LIN {X 18.143,Y -25.308,Z -49.954,A -90.000,B 90.000,C 0.000} C_DIS
LIN {X 18.670,Y -25.308,Z -49.551,A -90.000,B 90.000,C 0.000} C_DIS
LIN {X 18.953,Y -25.308,Z -49.343,A -90.000,B 90.000,C 0.000} C_DIS
LIN {X 19.482,Y -25.308,Z -48.976,A -90.000,B 90.000,C 0.000} C_DIS
LIN {X 19.664,Y -25.308,Z -48.848,A -90.000,B 90.000,C 0.000} C_DIS
LIN {X 20.308,Y -25.308,Z -48.429,A -90.000,B 90.000,C 0.000} C_DIS
LIN {X 20.824,Y -25.308,Z -48.139,A -90.000,B 90.000,C 0.000} C_DIS
LIN {X 21.214,Y -25.308,Z -47.885,A -90.000,B 90.000,C 0.000} C_DIS
LIN {X 21.722,Y -25.308,Z -47.610,A -90.000,B 90.000,C 0.000} C_DIS
LIN {X 22.049,Y -25.308,Z -47.442,A -90.000,B 90.000,C 0.000} C_DIS
LIN {X 22.838,Y -25.308,Z -47.072,A -90.000,B 90.000,C 0.000} C_DIS
LIN {X 23.297,Y -25.308,Z -46.836,A -90.000,B 90.000,C 0.000} C_DIS
LIN {X 23.748,Y -25.308,Z -46.617,A -90.000,B 90.000,C 0.000} C_DIS
LIN {X 24.114,Y -25.308,Z -46.450,A -90.000,B 90.000,C 0.000} C_DIS
LIN {X 24.501,Y -25.308,Z -46.297,A -90.000,B 90.000,C 0.000} C_DIS
LIN {X 25.566,Y -25.308,Z -45.827,A -90.000,B 90.000,C 0.000} C_DIS
LIN {X 26.230,Y -25.308,Z -45.591,A -90.000,B 90.000,C 0.000} C_DIS
LIN {X 26.539,Y -25.308,Z -45.462,A -90.000,B 90.000,C 0.000} C_DIS
LIN {X 27.063,Y -25.308,Z -45.267,A -90.000,B 90.000,C 0.000} C_DIS
LIN {X 27.873,Y -25.308,Z -45.015,A -90.000,B 90.000,C 0.000} C_DIS
LIN {X 28.137,Y -25.308,Z -44.933,A -90.000,B 90.000,C 0.000} C_DIS
LIN {X 28.312,Y -25.308,Z -44.875,A -90.000,B 90.000,C 0.000} C_DIS
LIN {X 28.933,Y -25.308,Z -44.707,A -90.000,B 90.000,C 0.000} C_DIS
LIN {X 29.591,Y -25.308,Z -44.529,A -90.000,B 90.000,C 0.000} C_DIS
LIN {X 30.404,Y -25.308,Z -44.390,A -90.000,B 90.000,C 0.000} C_DIS
LIN {X 30.883,Y -25.308,Z -44.298,A -90.000,B 90.000,C 0.000} C_DIS
LIN {X 31.361,Y -25.308,Z -44.231,A -90.000,B 90.000,C 0.000} C_DIS
LIN {X 31.445,Y -25.308,Z -44.222,A -90.000,B 90.000,C 0.000} C_DIS
LIN {X 31.957,Y -25.308,Z -44.139,A -90.000,B 90.000,C 0.000} C_DIS
LIN {X 32.533,Y -25.308,Z -44.081,A -90.000,B 90.000,C 0.000} C_DIS
LIN {X 32.602,Y -25.308,Z -44.069,A -90.000,B 90.000,C 0.000} C_DIS
LIN {X 33.150,Y -25.308,Z -43.994,A -90.000,B 90.000,C 0.000} C_DIS
LIN {X 33.474,Y -25.308,Z -43.910,A -90.000,B 90.000,C 0.000} C_DIS
LIN {X 34.801,Y -25.308,Z -43.463,A -90.000,B 90.000,C 0.000} C_DIS
LIN {X 36.507,Y -25.308,Z -42.820,A -90.000,B 90.000,C 0.000} C_DIS
LIN {X 38.163,Y -25.308,Z -42.257,A -90.000,B 90.000,C 0.000} C_DIS
LIN {X 38.421,Y -25.308,Z -42.166,A -90.000,B 90.000,C 0.000} C_DIS
LIN {X 38.842,Y -25.308,Z -42.036,A -90.000,B 90.000,C 0.000} C_DIS
LIN {X 38.933,Y -25.308,Z -42.009,A -90.000,B 90.000,C 0.000} C_DIS
LIN {X 40.215,Y -25.308,Z -41.708,A -90.000,B 90.000,C 0.000} C_DIS
LIN {X 40.698,Y -25.308,Z -41.598,A -90.000,B 90.000,C 0.000} C_DIS
LIN {X 41.808,Y -25.308,Z -41.425,A -90.000,B 90.000,C 0.000} C_DIS
LIN {X 42.260,Y -25.308,Z -41.365,A -90.000,B 90.000,C 0.000} C_DIS
LIN {X 42.548,Y -25.308,Z -41.331,A -90.000,B 90.000,C 0.000} C_DIS
LIN {X 42.938,Y -25.308,Z -41.302,A -90.000,B 90.000,C 0.000} C_DIS
LIN {X 43.127,Y -25.308,Z -41.298,A -90.000,B 90.000,C 0.000} C_DIS
LIN {X 44.357,Y -25.308,Z -41.301,A -90.000,B 90.000,C 0.000} C_DIS
LIN {X 44.824,Y -25.308,Z -41.310,A -90.000,B 90.000,C 0.000} C_DIS
LIN {X 46.077,Y -25.308,Z -41.438,A -90.000,B 90.000,C 0.000} C_DIS
LIN {X 46.591,Y -25.308,Z -41.498,A -90.000,B 90.000,C 0.000} C_DIS
LIN {X 46.783,Y -25.308,Z -41.522,A -90.000,B 90.000,C 0.000} C_DIS
LIN {X 47.059,Y -25.308,Z -41.565,A -90.000,B 90.000,C 0.000} C_DIS
LIN {X 47.466,Y -25.308,Z -41.664,A -90.000,B 90.000,C 0.000} C_DIS
LIN {X 47.871,Y -25.308,Z -41.771,A -90.000,B 90.000,C 0.000} C_DIS
LIN {X 49.147,Y -25.308,Z -42.145,A -90.000,B 90.000,C 0.000} C_DIS
LIN {X 50.476,Y -25.308,Z -42.617,A -90.000,B 90.000,C 0.000} C_DIS
LIN {X 50.921,Y -25.308,Z -42.786,A -90.000,B 90.000,C 0.000} C_DIS
LIN {X 51.227,Y -25.308,Z -42.923,A -90.000,B 90.000,C 0.000} C_DIS
LIN {X 52.706,Y -25.308,Z -43.641,A -90.000,B 90.000,C 0.000} C_DIS
LIN {X 53.133,Y -25.308,Z -43.865,A -90.000,B 90.000,C 0.000} C_DIS
LIN {X 53.694,Y -25.308,Z -44.165,A -90.000,B 90.000,C 0.000} C_DIS
LIN {X 54.079,Y -25.308,Z -44.378,A -90.000,B 90.000,C 0.000} C_DIS
LIN {X 54.481,Y -25.308,Z -44.646,A -90.000,B 90.000,C 0.000} C_DIS
LIN {X 55.761,Y -25.308,Z -45.510,A -90.000,B 90.000,C 0.000} C_DIS
LIN {X 56.981,Y -25.308,Z -46.342,A -90.000,B 90.000,C 0.000} C_DIS
LIN {X 57.354,Y -25.308,Z -46.650,A -90.000,B 90.000,C 0.000} C_DIS
LIN {X 59.159,Y -25.308,Z -48.157,A -90.000,B 90.000,C 0.000} C_DIS
LIN {X 59.556,Y -25.308,Z -48.497,A -90.000,B 90.000,C 0.000} C_DIS
LIN {X 61.541,Y -25.308,Z -50.392,A -90.000,B 90.000,C 0.000} C_DIS
LIN {X 62.293,Y -25.308,Z -51.104,A -90.000,B 90.000,C 0.000} C_DIS
LIN {X 63.430,Y -25.308,Z -52.202,A -90.000,B 90.000,C 0.000} C_DIS
LIN {X 64.564,Y -25.308,Z -53.172,A -90.000,B 90.000,C 0.000} C_DIS
LIN {X 65.147,Y -25.308,Z -53.687,A -90.000,B 90.000,C 0.000} C_DIS
LIN {X 65.829,Y -25.308,Z -54.185,A -90.000,B 90.000,C 0.000} C_DIS
LIN {X 67.069,Y -25.308,Z -55.053,A -90.000,B 90.000,C 0.000} C_DIS
LIN {X 67.323,Y -25.308,Z -55.221,A -90.000,B 90.000,C 0.000} C_DIS
LIN {X 68.793,Y -25.308,Z -56.153,A -90.000,B 90.000,C 0.000} C_DIS
LIN {X 69.363,Y -25.308,Z -56.519,A -90.000,B 90.000,C 0.000} C_DIS
LIN {X 70.905,Y -25.308,Z -57.502,A -90.000,B 90.000,C 0.000} C_DIS
LIN {X 71.252,Y -25.308,Z -57.727,A -90.000,B 90.000,C 0.000} C_DIS
LIN {X 71.570,Y -25.308,Z -57.963,A -90.000,B 90.000,C 0.000} C_DIS
LIN {X 73.123,Y -25.308,Z -59.076,A -90.000,B 90.000,C 0.000} C_DIS
LIN {X 73.494,Y -25.308,Z -59.375,A -90.000,B 90.000,C 0.000} C_DIS
LIN {X 74.370,Y -25.308,Z -60.174,A -90.000,B 90.000,C 0.000} C_DIS
LIN {X 75.025,Y -25.308,Z -60.802,A -90.000,B 90.000,C 0.000} C_DIS
LIN {X 75.362,Y -25.308,Z -61.138,A -90.000,B 90.000,C 0.000} C_DIS
LIN {X 75.788,Y -25.308,Z -61.621,A -90.000,B 90.000,C 0.000} C_DIS
LIN {X 76.413,Y -25.308,Z -62.367,A -90.000,B 90.000,C 0.000} C_DIS
LIN {X 76.829,Y -25.308,Z -62.865,A -90.000,B 90.000,C 0.000} C_DIS
LIN {X 77.271,Y -25.308,Z -63.464,A -90.000,B 90.000,C 0.000} C_DIS
LIN {X 77.867,Y -25.308,Z -64.321,A -90.000,B 90.000,C 0.000} C_DIS
LIN {X 78.264,Y -25.308,Z -64.917,A -90.000,B 90.000,C 0.000} C_DIS
LIN {X 78.540,Y -25.308,Z -65.359,A -90.000,B 90.000,C 0.000} C_DIS
LIN {X 79.035,Y -25.308,Z -63.677,A -90.000,B 90.000,C 0.000} C_DIS
LIN {X 79.744,Y -25.308,Z -61.550,A -90.000,B 90.000,C 0.000} C_DIS
LIN {X 79.787,Y -25.308,Z -61.436,A -90.000,B 90.000,C 0.000} C_DIS
LIN {X 80.298,Y -25.308,Z -59.798,A -90.000,B 90.000,C 0.000} C_DIS
LIN {X 80.453,Y -25.308,Z -59.335,A -90.000,B 90.000,C 0.000} C_DIS
LIN {X 81.205,Y -25.308,Z -57.294,A -90.000,B 90.000,C 0.000} C_DIS
LIN {X 81.746,Y -25.308,Z -56.077,A -90.000,B 90.000,C 0.000} C_DIS
LIN {X 82.134,Y -25.308,Z -55.110,A -90.000,B 90.000,C 0.000} C_DIS
LIN {X 82.335,Y -25.308,Z -54.666,A -90.000,B 90.000,C 0.000} C_DIS
LIN {X 83.333,Y -25.308,Z -52.807,A -90.000,B 90.000,C 0.000} C_DIS
LIN {X 83.579,Y -25.308,Z -52.386,A -90.000,B 90.000,C 0.000} C_DIS
LIN {X 84.744,Y -25.308,Z -50.676,A -90.000,B 90.000,C 0.000} C_DIS
LIN {X 85.030,Y -25.308,Z -50.284,A -90.000,B 90.000,C 0.000} C_DIS
LIN {X 86.347,Y -25.308,Z -48.703,A -90.000,B 90.000,C 0.000} C_DIS
LIN {X 86.674,Y -25.308,Z -48.341,A -90.000,B 90.000,C 0.000} C_DIS
LIN {X 88.117,Y -25.308,Z -46.880,A -90.000,B 90.000,C 0.000} C_DIS
LIN {X 88.495,Y -25.308,Z -46.539,A -90.000,B 90.000,C 0.000} C_DIS
LIN {X 90.061,Y -25.308,Z -45.164,A -90.000,B 90.000,C 0.000} C_DIS
LIN {X 91.724,Y -25.308,Z -43.871,A -90.000,B 90.000,C 0.000} C_DIS
LIN {X 92.141,Y -25.308,Z -43.566,A -90.000,B 90.000,C 0.000} C_DIS
LIN {X 93.780,Y -25.308,Z -42.419,A -90.000,B 90.000,C 0.000} C_DIS
LIN {X 95.430,Y -25.308,Z -41.375,A -90.000,B 90.000,C 0.000} C_DIS
LIN {X 95.885,Y -25.308,Z -41.109,A -90.000,B 90.000,C 0.000} C_DIS
LIN {X 97.376,Y -25.308,Z -40.260,A -90.000,B 90.000,C 0.000} C_DIS
LIN {X 98.805,Y -25.308,Z -39.523,A -90.000,B 90.000,C 0.000} C_DIS
LIN {X 100.339,Y -25.308,Z -38.797,A -90.000,B 90.000,C 0.000} C_DIS
LIN {X 102.099,Y -25.308,Z -37.999,A -90.000,B 90.000,C 0.000} C_DIS
LIN {X 103.528,Y -25.308,Z -37.362,A -90.000,B 90.000,C 0.000} C_DIS
LIN {X 104.529,Y -25.308,Z -36.920,A -90.000,B 90.000,C 0.000} C_DIS
LIN {X 105.418,Y -25.308,Z -36.546,A -90.000,B 90.000,C 0.000} C_DIS
LIN {X 106.878,Y -25.308,Z -35.966,A -90.000,B 90.000,C 0.000} C_DIS
LIN {X 107.402,Y -25.308,Z -35.767,A -90.000,B 90.000,C 0.000} C_DIS
LIN {X 107.855,Y -25.308,Z -35.604,A -90.000,B 90.000,C 0.000} C_DIS
LIN {X 108.317,Y -25.308,Z -35.448,A -90.000,B 90.000,C 0.000} C_DIS
LIN {X 108.777,Y -25.308,Z -35.326,A -90.000,B 90.000,C 0.000} C_DIS
LIN {X 109.221,Y -25.308,Z -35.225,A -90.000,B 90.000,C 0.000} C_DIS
LIN {X 109.760,Y -25.308,Z -35.155,A -90.000,B 90.000,C 0.000} C_DIS
LIN {X 110.108,Y -25.308,Z -35.113,A -90.000,B 90.000,C 0.000} C_DIS
LIN {X 110.563,Y -25.308,Z -35.105,A -90.000,B 90.000,C 0.000} C_DIS
LIN {X 110.619,Y -25.308,Z -35.106,A -90.000,B 90.000,C 0.000} C_DIS
LIN {X 110.949,Y -25.308,Z -35.117,A -90.000,B 90.000,C 0.000} C_DIS
LIN {X 111.445,Y -25.308,Z -35.160,A -90.000,B 90.000,C 0.000} C_DIS
LIN {X 112.068,Y -25.308,Z -35.277,A -90.000,B 90.000,C 0.000} C_DIS
LIN {X 112.405,Y -25.308,Z -35.362,A -90.000,B 90.000,C 0.000} C_DIS
LIN {X 112.925,Y -25.308,Z -35.518,A -90.000,B 90.000,C 0.000} C_DIS
LIN {X 113.055,Y -25.308,Z -35.560,A -90.000,B 90.000,C 0.000} C_DIS
LIN {X 113.505,Y -25.308,Z -35.746,A -90.000,B 90.000,C 0.000} C_DIS
LIN {X 113.979,Y -25.308,Z -35.973,A -90.000,B 90.000,C 0.000} C_DIS
LIN {X 114.418,Y -25.308,Z -36.210,A -90.000,B 90.000,C 0.000} C_DIS
LIN {X 114.540,Y -25.308,Z -36.286,A -90.000,B 90.000,C 0.000} C_DIS
LIN {X 114.952,Y -25.308,Z -36.566,A -90.000,B 90.000,C 0.000} C_DIS
LIN {X 115.050,Y -25.308,Z -36.644,A -90.000,B 90.000,C 0.000} C_DIS
LIN {X 115.450,Y -25.308,Z -36.982,A -90.000,B 90.000,C 0.000} C_DIS
LIN {X 115.513,Y -25.308,Z -37.039,A -90.000,B 90.000,C 0.000} C_DIS
LIN {X 115.921,Y -25.308,Z -37.462,A -90.000,B 90.000,C 0.000} C_DIS
LIN {X 116.080,Y -25.308,Z -37.632,A -90.000,B 90.000,C 0.000} C_DIS
LIN {X 116.439,Y -25.308,Z -38.088,A -90.000,B 90.000,C 0.000} C_DIS
LIN {X 116.700,Y -25.308,Z -38.500,A -90.000,B 90.000,C 0.000} C_DIS
LIN {X 116.928,Y -25.308,Z -38.961,A -90.000,B 90.000,C 0.000} C_DIS
LIN {X 117.066,Y -25.308,Z -39.268,A -90.000,B 90.000,C 0.000} C_DIS
LIN {X 117.142,Y -25.308,Z -39.466,A -90.000,B 90.000,C 0.000} C_DIS
LIN {X 117.260,Y -25.308,Z -39.781,A -90.000,B 90.000,C 0.000} C_DIS
LIN {X 117.390,Y -25.308,Z -40.280,A -90.000,B 90.000,C 0.000} C_DIS
LIN {X 117.462,Y -25.308,Z -40.593,A -90.000,B 90.000,C 0.000} C_DIS
LIN {X 117.541,Y -25.308,Z -41.107,A -90.000,B 90.000,C 0.000} C_DIS
LIN {X 117.596,Y -25.308,Z -41.523,A -90.000,B 90.000,C 0.000} C_DIS
LIN {X 117.630,Y -25.308,Z -41.874,A -90.000,B 90.000,C 0.000} C_DIS
LIN {X 117.659,Y -25.308,Z -42.461,A -90.000,B 90.000,C 0.000} C_DIS
LIN {X 117.668,Y -25.308,Z -42.696,A -90.000,B 90.000,C 0.000} C_DIS
LIN {X 117.664,Y -25.308,Z -42.866,A -90.000,B 90.000,C 0.000} C_DIS
LIN {X 117.661,Y -25.308,Z -42.950,A -90.000,B 90.000,C 0.000} C_DIS
LIN {X 117.651,Y -25.308,Z -43.202,A -90.000,B 90.000,C 0.000} C_DIS
LIN {X 117.607,Y -25.308,Z -43.721,A -90.000,B 90.000,C 0.000} C_DIS
LIN {X 117.567,Y -25.308,Z -44.117,A -90.000,B 90.000,C 0.000} C_DIS
LIN {X 117.482,Y -25.308,Z -44.670,A -90.000,B 90.000,C 0.000} C_DIS
LIN {X 117.399,Y -25.308,Z -45.114,A -90.000,B 90.000,C 0.000} C_DIS
LIN {X 117.260,Y -25.308,Z -45.739,A -90.000,B 90.000,C 0.000} C_DIS
LIN {X 117.105,Y -25.308,Z -46.261,A -90.000,B 90.000,C 0.000} C_DIS
LIN {X 116.900,Y -25.308,Z -46.938,A -90.000,B 90.000,C 0.000} C_DIS
LIN {X 116.546,Y -25.308,Z -47.857,A -90.000,B 90.000,C 0.000} C_DIS
LIN {X 116.372,Y -25.308,Z -48.278,A -90.000,B 90.000,C 0.000} C_DIS
LIN {X 115.873,Y -25.308,Z -49.350,A -90.000,B 90.000,C 0.000} C_DIS
LIN {X 115.235,Y -25.308,Z -50.626,A -90.000,B 90.000,C 0.000} C_DIS
LIN {X 114.577,Y -25.308,Z -51.931,A -90.000,B 90.000,C 0.000} C_DIS
LIN {X 113.941,Y -25.308,Z -53.229,A -90.000,B 90.000,C 0.000} C_DIS
LIN {X 113.276,Y -25.308,Z -54.687,A -90.000,B 90.000,C 0.000} C_DIS
LIN {X 112.799,Y -25.308,Z -55.830,A -90.000,B 90.000,C 0.000} C_DIS
LIN {X 112.213,Y -25.308,Z -57.388,A -90.000,B 90.000,C 0.000} C_DIS
LIN {X 111.674,Y -25.308,Z -59.009,A -90.000,B 90.000,C 0.000} C_DIS
LIN {X 111.260,Y -25.308,Z -60.445,A -90.000,B 90.000,C 0.000} C_DIS
LIN {X 110.703,Y -25.308,Z -62.486,A -90.000,B 90.000,C 0.000} C_DIS
LIN {X 110.152,Y -25.308,Z -64.437,A -90.000,B 90.000,C 0.000} C_DIS
LIN {X 110.021,Y -25.308,Z -64.879,A -90.000,B 90.000,C 0.000} C_DIS
LIN {X 109.345,Y -25.308,Z -67.050,A -90.000,B 90.000,C 0.000} C_DIS
LIN {X 108.519,Y -25.308,Z -69.358,A -90.000,B 90.000,C 0.000} C_DIS
LIN {X 107.550,Y -25.308,Z -71.793,A -90.000,B 90.000,C 0.000} C_DIS
LIN {X 107.403,Y -25.308,Z -72.150,A -90.000,B 90.000,C 0.000} C_DIS
LIN {X 106.414,Y -25.308,Z -74.420,A -90.000,B 90.000,C 0.000} C_DIS
LIN {X 105.411,Y -25.308,Z -76.516,A -90.000,B 90.000,C 0.000} C_DIS
LIN {X 104.209,Y -25.308,Z -78.763,A -90.000,B 90.000,C 0.000} C_DIS
LIN {X 103.943,Y -25.308,Z -79.223,A -90.000,B 90.000,C 0.000} C_DIS
LIN {X 103.058,Y -25.308,Z -80.726,A -90.000,B 90.000,C 0.000} C_DIS
LIN {X 102.880,Y -25.308,Z -81.006,A -90.000,B 90.000,C 0.000} C_DIS
LIN {X 102.164,Y -25.308,Z -82.128,A -90.000,B 90.000,C 0.000} C_DIS
LIN {X 99.737,Y -25.308,Z -85.762,A -90.000,B 90.000,C 0.000} C_DIS
LIN {X 99.776,Y -25.308,Z -86.269,A -90.000,B 90.000,C 0.000} C_DIS
LIN {X 99.848,Y -25.308,Z -87.593,A -90.000,B 90.000,C 0.000} C_DIS
LIN {X 99.953,Y -25.308,Z -88.797,A -90.000,B 90.000,C 0.000} C_DIS
LIN {X 99.978,Y -25.308,Z -89.273,A -90.000,B 90.000,C 0.000} C_DIS
LIN {X 99.997,Y -25.308,Z -89.800,A -90.000,B 90.000,C 0.000} C_DIS
LIN {X 100.015,Y -25.308,Z -90.712,A -90.000,B 90.000,C 0.000} C_DIS
LIN {X 100.028,Y -25.308,Z -91.629,A -90.000,B 90.000,C 0.000} C_DIS
LIN {X 100.042,Y -25.308,Z -92.081,A -90.000,B 90.000,C 0.000} C_DIS
LIN {X 100.041,Y -25.308,Z -92.155,A -90.000,B 90.000,C 0.000} C_DIS
LIN {X 99.990,Y -25.308,Z -93.020,A -90.000,B 90.000,C 0.000} C_DIS
LIN {X 99.954,Y -25.308,Z -93.959,A -90.000,B 90.000,C 0.000} C_DIS
LIN {X 99.931,Y -25.308,Z -94.384,A -90.000,B 90.000,C 0.000} C_DIS
LIN {X 99.913,Y -25.308,Z -94.531,A -90.000,B 90.000,C 0.000} C_DIS
LIN {X 99.819,Y -25.308,Z -95.415,A -90.000,B 90.000,C 0.000} C_DIS
LIN {X 99.799,Y -25.308,Z -95.920,A -90.000,B 90.000,C 0.000} C_DIS
LIN {X 99.741,Y -25.308,Z -96.399,A -90.000,B 90.000,C 0.000} C_DIS
LIN {X 99.696,Y -25.308,Z -96.658,A -90.000,B 90.000,C 0.000} C_DIS
LIN {X 99.644,Y -25.308,Z -97.627,A -90.000,B 90.000,C 0.000} C_DIS
LIN {X 99.544,Y -25.308,Z -99.179,A -90.000,B 90.000,C 0.000} C_DIS
LIN {X 99.527,Y -25.308,Z -99.300,A -90.000,B 90.000,C 0.000} C_DIS
LIN {X 99.435,Y -25.308,Z -100.699,A -90.000,B 90.000,C 0.000} C_DIS
LIN {X 99.398,Y -25.308,Z -100.988,A -90.000,B 90.000,C 0.000} C_DIS
LIN {X 99.340,Y -25.308,Z -102.329,A -90.000,B 90.000,C 0.000} C_DIS
LIN {X 99.327,Y -25.308,Z -102.468,A -90.000,B 90.000,C 0.000} C_DIS
LIN {X 99.324,Y -25.308,Z -103.358,A -90.000,B 90.000,C 0.000} C_DIS
LIN {X 99.312,Y -25.308,Z -103.683,A -90.000,B 90.000,C 0.000} C_DIS
LIN {X 99.307,Y -25.308,Z -103.795,A -90.000,B 90.000,C 0.000} C_DIS
LIN {X 99.321,Y -25.308,Z -104.026,A -90.000,B 90.000,C 0.000} C_DIS
LIN {X 99.361,Y -25.308,Z -104.573,A -90.000,B 90.000,C 0.000} C_DIS
LIN {X 99.427,Y -25.308,Z -105.073,A -90.000,B 90.000,C 0.000} C_DIS
LIN {X 99.488,Y -25.308,Z -105.508,A -90.000,B 90.000,C 0.000} C_DIS
LIN {X 99.631,Y -25.308,Z -106.321,A -90.000,B 90.000,C 0.000} C_DIS
LIN {X 99.899,Y -25.308,Z -107.995,A -90.000,B 90.000,C 0.000} C_DIS
LIN {X 99.981,Y -25.308,Z -108.804,A -90.000,B 90.000,C 0.000} C_DIS
LIN {X 100.053,Y -25.308,Z -109.443,A -90.000,B 90.000,C 0.000} C_DIS
LIN {X 100.126,Y -25.308,Z -110.453,A -90.000,B 90.000,C 0.000} C_DIS
LIN {X 100.183,Y -25.308,Z -111.111,A -90.000,B 90.000,C 0.000} C_DIS
LIN {X 100.229,Y -25.308,Z -111.892,A -90.000,B 90.000,C 0.000} C_DIS
LIN {X 100.310,Y -25.308,Z -112.963,A -90.000,B 90.000,C 0.000} C_DIS
LIN {X 100.359,Y -25.308,Z -113.831,A -90.000,B 90.000,C 0.000} C_DIS
LIN {X 100.445,Y -25.308,Z -115.019,A -90.000,B 90.000,C 0.000} C_DIS
LIN {X 100.533,Y -25.308,Z -116.130,A -90.000,B 90.000,C 0.000} C_DIS
LIN {X 100.601,Y -25.308,Z -117.246,A -90.000,B 90.000,C 0.000} C_DIS
LIN {X 100.674,Y -25.308,Z -118.213,A -90.000,B 90.000,C 0.000} C_DIS
LIN {X 100.751,Y -25.308,Z -119.583,A -90.000,B 90.000,C 0.000} C_DIS
LIN {X 100.800,Y -25.308,Z -120.356,A -90.000,B 90.000,C 0.000} C_DIS
LIN {X 100.825,Y -25.308,Z -120.811,A -90.000,B 90.000,C 0.000} C_DIS
LIN {X 100.921,Y -25.308,Z -122.978,A -90.000,B 90.000,C 0.000} C_DIS
LIN {X 100.945,Y -25.308,Z -123.620,A -90.000,B 90.000,C 0.000} C_DIS
LIN {X 100.973,Y -25.308,Z -124.815,A -90.000,B 90.000,C 0.000} C_DIS
LIN {X 100.968,Y -25.308,Z -126.202,A -90.000,B 90.000,C 0.000} C_DIS
LIN {X 100.978,Y -25.308,Z -127.131,A -90.000,B 90.000,C 0.000} C_DIS
LIN {X 100.927,Y -25.308,Z -128.864,A -90.000,B 90.000,C 0.000} C_DIS
LIN {X 100.912,Y -25.308,Z -129.693,A -90.000,B 90.000,C 0.000} C_DIS
LIN {X 100.815,Y -25.308,Z -131.616,A -90.000,B 90.000,C 0.000} C_DIS
LIN {X 100.792,Y -25.308,Z -132.231,A -90.000,B 90.000,C 0.000} C_DIS
LIN {X 100.655,Y -25.308,Z -134.453,A -90.000,B 90.000,C 0.000} C_DIS
LIN {X 100.615,Y -25.308,Z -135.207,A -90.000,B 90.000,C 0.000} C_DIS
LIN {X 100.584,Y -25.308,Z -135.733,A -90.000,B 90.000,C 0.000} C_DIS
LIN {X 100.370,Y -25.308,Z -138.988,A -90.000,B 90.000,C 0.000} C_DIS
LIN {X 100.175,Y -25.308,Z -141.689,A -90.000,B 90.000,C 0.000} C_DIS
LIN {X 100.021,Y -25.308,Z -143.726,A -90.000,B 90.000,C 0.000} C_DIS
LIN {X 99.864,Y -25.308,Z -145.627,A -90.000,B 90.000,C 0.000} C_DIS
LIN {X 99.651,Y -25.308,Z -148.108,A -90.000,B 90.000,C 0.000} C_DIS
LIN {X 99.528,Y -25.308,Z -149.393,A -90.000,B 90.000,C 0.000} C_DIS
LIN {X 99.410,Y -25.308,Z -150.436,A -90.000,B 90.000,C 0.000} C_DIS
LIN {X 99.155,Y -25.308,Z -153.045,A -90.000,B 90.000,C 0.000} C_DIS
LIN {X 99.077,Y -25.308,Z -153.644,A -90.000,B 90.000,C 0.000} C_DIS
LIN {X 99.058,Y -25.308,Z -153.783,A -90.000,B 90.000,C 0.000} C_DIS
LIN {X 98.742,Y -25.308,Z -156.680,A -90.000,B 90.000,C 0.000} C_DIS
LIN {X 98.709,Y -25.308,Z -156.898,A -90.000,B 90.000,C 0.000} C_DIS
LIN {X 98.400,Y -25.308,Z -159.435,A -90.000,B 90.000,C 0.000} C_DIS
LIN {X 98.332,Y -25.308,Z -160.140,A -90.000,B 90.000,C 0.000} C_DIS
LIN {X 98.002,Y -25.308,Z -162.603,A -90.000,B 90.000,C 0.000} C_DIS
LIN {X 97.876,Y -25.308,Z -163.832,A -90.000,B 90.000,C 0.000} C_DIS
LIN {X 97.601,Y -25.308,Z -165.718,A -90.000,B 90.000,C 0.000} C_DIS
LIN {X 97.397,Y -25.308,Z -167.595,A -90.000,B 90.000,C 0.000} C_DIS
LIN {X 97.263,Y -25.308,Z -168.464,A -90.000,B 90.000,C 0.000} C_DIS
LIN {X 96.949,Y -25.308,Z -171.253,A -90.000,B 90.000,C 0.000} C_DIS
LIN {X 96.874,Y -25.308,Z -171.737,A -90.000,B 90.000,C 0.000} C_DIS
LIN {X 96.488,Y -25.308,Z -175.168,A -90.000,B 90.000,C 0.000} C_DIS
LIN {X 96.182,Y -25.308,Z -177.661,A -90.000,B 90.000,C 0.000} C_DIS
LIN {X 96.152,Y -25.308,Z -177.991,A -90.000,B 90.000,C 0.000} C_DIS
LIN {X 95.896,Y -25.308,Z -180.202,A -90.000,B 90.000,C 0.000} C_DIS
LIN {X 95.835,Y -25.308,Z -180.892,A -90.000,B 90.000,C 0.000} C_DIS
LIN {X 95.662,Y -25.308,Z -182.520,A -90.000,B 90.000,C 0.000} C_DIS
LIN {X 95.576,Y -25.308,Z -183.541,A -90.000,B 90.000,C 0.000} C_DIS
LIN {X 95.467,Y -25.308,Z -184.688,A -90.000,B 90.000,C 0.000} C_DIS
LIN {X 95.336,Y -25.308,Z -186.329,A -90.000,B 90.000,C 0.000} C_DIS
LIN {X 95.306,Y -25.308,Z -186.689,A -90.000,B 90.000,C 0.000} C_DIS
LIN {X 95.191,Y -25.308,Z -188.281,A -90.000,B 90.000,C 0.000} C_DIS
LIN {X 95.023,Y -25.308,Z -190.814,A -90.000,B 90.000,C 0.000} C_DIS
LIN {X 95.011,Y -25.308,Z -190.963,A -90.000,B 90.000,C 0.000} C_DIS
LIN {X 94.740,Y -25.308,Z -193.398,A -90.000,B 90.000,C 0.000} C_DIS
LIN {X 94.454,Y -25.308,Z -195.346,A -90.000,B 90.000,C 0.000} C_DIS
LIN {X 94.234,Y -25.308,Z -196.731,A -90.000,B 90.000,C 0.000} C_DIS
LIN {X 93.663,Y -25.308,Z -199.595,A -90.000,B 90.000,C 0.000} C_DIS
LIN {X 93.542,Y -25.308,Z -200.212,A -90.000,B 90.000,C 0.000} C_DIS
LIN {X 92.828,Y -25.308,Z -203.214,A -90.000,B 90.000,C 0.000} C_DIS
LIN {X 92.544,Y -25.308,Z -204.440,A -90.000,B 90.000,C 0.000} C_DIS
LIN {X 91.801,Y -25.308,Z -207.333,A -90.000,B 90.000,C 0.000} C_DIS
LIN {X 91.325,Y -25.308,Z -209.244,A -90.000,B 90.000,C 0.000} C_DIS
LIN {X 90.642,Y -25.308,Z -211.832,A -90.000,B 90.000,C 0.000} C_DIS
LIN {X 89.972,Y -25.308,Z -214.447,A -90.000,B 90.000,C 0.000} C_DIS
LIN {X 89.411,Y -25.308,Z -216.578,A -90.000,B 90.000,C 0.000} C_DIS
LIN {X 88.171,Y -25.308,Z -221.432,A -90.000,B 90.000,C 0.000} C_DIS
LIN {X 87.204,Y -25.308,Z -225.322,A -90.000,B 90.000,C 0.000} C_DIS
LIN {X 86.940,Y -25.308,Z -226.315,A -90.000,B 90.000,C 0.000} C_DIS
LIN {X 85.743,Y -25.308,Z -230.924,A -90.000,B 90.000,C 0.000} C_DIS
LIN {X 85.646,Y -25.308,Z -231.281,A -90.000,B 90.000,C 0.000} C_DIS
LIN {X 85.522,Y -25.308,Z -231.698,A -90.000,B 90.000,C 0.000} C_DIS
LIN {X 84.416,Y -25.308,Z -235.552,A -90.000,B 90.000,C 0.000} C_DIS
LIN {X 83.986,Y -25.308,Z -237.019,A -90.000,B 90.000,C 0.000} C_DIS
LIN {X 81.908,Y -25.308,Z -243.223,A -90.000,B 90.000,C 0.000} C_DIS
LIN {X 81.778,Y -25.308,Z -243.561,A -90.000,B 90.000,C 0.000} C_DIS
LIN {X 81.778,Y -60.000,Z -243.561,A -90.000,B 90.000,C 0.000} C_DIS
LIN {X 99.796,Y -60.000,Z -86.519,A -90.000,B 90.000,C 0.000} C_DIS
LIN {X 99.796,Y -23.308,Z -86.519,A -90.000,B 90.000,C 0.000} C_DIS
LIN {X 99.871,Y -23.309,Z -87.492,A -90.000,B 90.000,C 0.000} C_DIS
LIN {X 100.033,Y -23.309,Z -89.800,A -90.000,B 90.000,C 0.000} C_DIS
LIN {X 100.049,Y -23.309,Z -90.038,A -90.000,B 90.000,C 0.000} C_DIS
LIN {X 100.093,Y -23.310,Z -90.499,A -90.000,B 90.000,C 0.000} C_DIS
LIN {X 100.109,Y -23.311,Z -90.717,A -90.000,B 90.000,C 0.000} C_DIS
LIN {X 100.173,Y -23.313,Z -91.776,A -90.000,B 90.000,C 0.000} C_DIS
LIN {X 100.205,Y -23.315,Z -92.181,A -90.000,B 90.000,C 0.000} C_DIS
LIN {X 100.234,Y -23.319,Z -92.418,A -90.000,B 90.000,C 0.000} C_DIS
LIN {X 100.259,Y -23.326,Z -92.902,A -90.000,B 90.000,C 0.000} C_DIS
LIN {X 100.244,Y -23.328,Z -93.631,A -90.000,B 90.000,C 0.000} C_DIS
LIN {X 100.269,Y -23.339,Z -94.490,A -90.000,B 90.000,C 0.000} C_DIS
LIN {X 100.271,Y -23.340,Z -94.538,A -90.000,B 90.000,C 0.000} C_DIS
LIN {X 100.259,Y -23.345,Z -94.860,A -90.000,B 90.000,C 0.000} C_DIS
LIN {X 100.222,Y -23.350,Z -95.541,A -90.000,B 90.000,C 0.000} C_DIS
LIN {X 100.217,Y -23.350,Z -95.646,A -90.000,B 90.000,C 0.000} C_DIS
LIN {X 100.224,Y -23.354,Z -95.935,A -90.000,B 90.000,C 0.000} C_DIS
LIN {X 100.212,Y -23.360,Z -96.257,A -90.000,B 90.000,C 0.000} C_DIS
LIN {X 100.177,Y -23.368,Z -96.708,A -90.000,B 90.000,C 0.000} C_DIS
LIN {X 100.162,Y -23.367,Z -96.923,A -90.000,B 90.000,C 0.000} C_DIS
LIN {X 100.162,Y -23.367,Z -96.956,A -90.000,B 90.000,C 0.000} C_DIS
LIN {X 100.164,Y -23.387,Z -98.180,A -90.000,B 90.000,C 0.000} C_DIS
LIN {X 100.163,Y -23.389,Z -98.333,A -90.000,B 90.000,C 0.000} C_DIS
LIN {X 100.144,Y -23.391,Z -98.741,A -90.000,B 90.000,C 0.000} C_DIS
LIN {X 100.124,Y -23.391,Z -99.045,A -90.000,B 90.000,C 0.000} C_DIS
LIN {X 100.126,Y -23.398,Z -99.275,A -90.000,B 90.000,C 0.000} C_DIS
LIN {X 100.129,Y -23.412,Z -99.834,A -90.000,B 90.000,C 0.000} C_DIS
LIN {X 100.110,Y -23.415,Z -100.241,A -90.000,B 90.000,C 0.000} C_DIS
LIN {X 100.081,Y -23.415,Z -100.672,A -90.000,B 90.000,C 0.000} C_DIS
LIN {X 100.086,Y -23.431,Z -101.042,A -90.000,B 90.000,C 0.000} C_DIS
LIN {X 100.092,Y -23.437,Z -101.310,A -90.000,B 90.000,C 0.000} C_DIS
LIN {X 100.065,Y -23.439,Z -102.005,A -90.000,B 90.000,C 0.000} C_DIS
LIN {X 100.057,Y -23.439,Z -102.203,A -90.000,B 90.000,C 0.000} C_DIS
LIN {X 100.069,Y -23.452,Z -102.533,A -90.000,B 90.000,C 0.000} C_DIS
LIN {X 100.088,Y -23.460,Z -102.959,A -90.000,B 90.000,C 0.000} C_DIS
LIN {X 100.086,Y -23.461,Z -103.455,A -90.000,B 90.000,C 0.000} C_DIS
LIN {X 100.086,Y -23.462,Z -103.545,A -90.000,B 90.000,C 0.000} C_DIS
LIN {X 100.103,Y -23.472,Z -103.832,A -90.000,B 90.000,C 0.000} C_DIS
LIN {X 100.116,Y -23.473,Z -103.986,A -90.000,B 90.000,C 0.000} C_DIS
LIN {X 100.166,Y -23.480,Z -104.480,A -90.000,B 90.000,C 0.000} C_DIS
LIN {X 100.256,Y -23.482,Z -105.112,A -90.000,B 90.000,C 0.000} C_DIS
LIN {X 100.300,Y -23.484,Z -105.388,A -90.000,B 90.000,C 0.000} C_DIS
LIN {X 100.456,Y -23.485,Z -106.279,A -90.000,B 90.000,C 0.000} C_DIS
LIN {X 100.723,Y -23.487,Z -107.938,A -90.000,B 90.000,C 0.000} C_DIS
LIN {X 100.802,Y -23.490,Z -108.638,A -90.000,B 90.000,C 0.000} C_DIS
LIN {X 100.889,Y -23.493,Z -109.358,A -90.000,B 90.000,C 0.000} C_DIS
LIN {X 100.940,Y -23.497,Z -109.957,A -90.000,B 90.000,C 0.000} C_DIS
LIN {X 101.003,Y -23.503,Z -110.603,A -90.000,B 90.000,C 0.000} C_DIS
LIN {X 101.045,Y -23.505,Z -111.036,A -90.000,B 90.000,C 0.000} C_DIS
LIN {X 101.096,Y -23.510,Z -111.725,A -90.000,B 90.000,C 0.000} C_DIS
LIN {X 101.200,Y -23.519,Z -112.897,A -90.000,B 90.000,C 0.000} C_DIS
LIN {X 101.226,Y -23.521,Z -113.263,A -90.000,B 90.000,C 0.000} C_DIS
LIN {X 101.275,Y -23.529,Z -113.835,A -90.000,B 90.000,C 0.000} C_DIS
LIN {X 101.376,Y -23.539,Z -114.970,A -90.000,B 90.000,C 0.000} C_DIS
LIN {X 101.480,Y -23.548,Z -116.073,A -90.000,B 90.000,C 0.000} C_DIS
LIN {X 101.526,Y -23.556,Z -116.584,A -90.000,B 90.000,C 0.000} C_DIS
LIN {X 101.573,Y -23.561,Z -117.187,A -90.000,B 90.000,C 0.000} C_DIS
LIN {X 101.660,Y -23.569,Z -118.158,A -90.000,B 90.000,C 0.000} C_DIS
LIN {X 101.706,Y -23.578,Z -118.699,A -90.000,B 90.000,C 0.000} C_DIS
LIN {X 101.772,Y -23.586,Z -119.630,A -90.000,B 90.000,C 0.000} C_DIS
LIN {X 101.859,Y -23.597,Z -120.765,A -90.000,B 90.000,C 0.000} C_DIS
LIN {X 101.866,Y -23.598,Z -120.866,A -90.000,B 90.000,C 0.000} C_DIS
LIN {X 101.990,Y -23.616,Z -123.057,A -90.000,B 90.000,C 0.000} C_DIS
LIN {X 102.019,Y -23.621,Z -123.660,A -90.000,B 90.000,C 0.000} C_DIS
LIN {X 102.043,Y -23.628,Z -124.189,A -90.000,B 90.000,C 0.000} C_DIS
LIN {X 102.063,Y -23.632,Z -124.772,A -90.000,B 90.000,C 0.000} C_DIS
LIN {X 102.069,Y -23.637,Z -125.462,A -90.000,B 90.000,C 0.000} C_DIS
LIN {X 102.085,Y -23.649,Z -126.246,A -90.000,B 90.000,C 0.000} C_DIS
LIN {X 102.105,Y -23.656,Z -127.118,A -90.000,B 90.000,C 0.000} C_DIS
LIN {X 102.087,Y -23.663,Z -128.074,A -90.000,B 90.000,C 0.000} C_DIS
LIN {X 102.079,Y -23.675,Z -128.939,A -90.000,B 90.000,C 0.000} C_DIS
LIN {X 102.076,Y -23.680,Z -129.516,A -90.000,B 90.000,C 0.000} C_DIS
LIN {X 102.072,Y -23.679,Z -129.714,A -90.000,B 90.000,C 0.000} C_DIS
LIN {X 102.023,Y -23.686,Z -130.895,A -90.000,B 90.000,C 0.000} C_DIS
LIN {X 101.998,Y -23.696,Z -131.668,A -90.000,B 90.000,C 0.000} C_DIS
LIN {X 101.981,Y -23.700,Z -132.276,A -90.000,B 90.000,C 0.000} C_DIS
LIN {X 101.900,Y -23.707,Z -133.748,A -90.000,B 90.000,C 0.000} C_DIS
LIN {X 101.860,Y -23.715,Z -134.583,A -90.000,B 90.000,C 0.000} C_DIS
LIN {X 101.834,Y -23.718,Z -135.142,A -90.000,B 90.000,C 0.000} C_DIS
LIN {X 101.801,Y -23.721,Z -135.769,A -90.000,B 90.000,C 0.000} C_DIS
LIN {X 101.734,Y -23.728,Z -136.925,A -90.000,B 90.000,C 0.000} C_DIS
LIN {X 101.602,Y -23.735,Z -139.077,A -90.000,B 90.000,C 0.000} C_DIS
LIN {X 101.466,Y -23.747,Z -141.169,A -90.000,B 90.000,C 0.000} C_DIS
LIN {X 101.288,Y -23.757,Z -143.708,A -90.000,B 90.000,C 0.000} C_DIS
LIN {X 101.206,Y -23.764,Z -144.816,A -90.000,B 90.000,C 0.000} C_DIS
LIN {X 101.027,Y -23.774,Z -147.084,A -90.000,B 90.000,C 0.000} C_DIS
LIN {X 100.935,Y -23.780,Z -148.230,A -90.000,B 90.000,C 0.000} C_DIS
LIN {X 100.906,Y -23.783,Z -148.576,A -90.000,B 90.000,C 0.000} C_DIS
LIN {X 100.822,Y -23.788,Z -149.521,A -90.000,B 90.000,C 0.000} C_DIS
LIN {X 100.786,Y -23.791,Z -149.864,A -90.000,B 90.000,C 0.000} C_DIS
LIN {X 100.718,Y -23.801,Z -150.578,A -90.000,B 90.000,C 0.000} C_DIS
LIN {X 100.482,Y -23.820,Z -153.205,A -90.000,B 90.000,C 0.000} C_DIS
LIN {X 100.461,Y -23.822,Z -153.380,A -90.000,B 90.000,C 0.000} C_DIS
LIN {X 100.399,Y -23.833,Z -153.945,A -90.000,B 90.000,C 0.000} C_DIS
LIN {X 100.219,Y -23.851,Z -155.774,A -90.000,B 90.000,C 0.000} C_DIS
LIN {X 100.107,Y -23.861,Z -156.883,A -90.000,B 90.000,C 0.000} C_DIS
LIN {X 100.083,Y -23.866,Z -157.084,A -90.000,B 90.000,C 0.000} C_DIS
LIN {X 99.804,Y -23.892,Z -159.588,A -90.000,B 90.000,C 0.000} C_DIS
LIN {X 99.750,Y -23.892,Z -160.145,A -90.000,B 90.000,C 0.000} C_DIS
LIN {X 99.733,Y -23.893,Z -160.328,A -90.000,B 90.000,C 0.000} C_DIS
LIN {X 99.704,Y -23.899,Z -160.591,A -90.000,B 90.000,C 0.000} C_DIS
LIN {X 99.439,Y -23.928,Z -162.772,A -90.000,B 90.000,C 0.000} C_DIS
LIN {X 99.320,Y -23.941,Z -164.043,A -90.000,B 90.000,C 0.000} C_DIS
LIN {X 99.079,Y -23.969,Z -165.878,A -90.000,B 90.000,C 0.000} C_DIS
LIN {X 98.892,Y -23.990,Z -167.756,A -90.000,B 90.000,C 0.000} C_DIS
LIN {X 98.766,Y -24.003,Z -168.664,A -90.000,B 90.000,C 0.000} C_DIS
LIN {X 98.705,Y -24.001,Z -169.186,A -90.000,B 90.000,C 0.000} C_DIS
LIN {X 98.474,Y -24.026,Z -171.421,A -90.000,B 90.000,C 0.000} C_DIS
LIN {X 98.426,Y -24.030,Z -171.768,A -90.000,B 90.000,C 0.000} C_DIS
LIN {X 98.404,Y -24.035,Z -171.940,A -90.000,B 90.000,C 0.000} C_DIS
LIN {X 98.101,Y -24.064,Z -174.841,A -90.000,B 90.000,C 0.000} C_DIS
LIN {X 98.041,Y -24.069,Z -175.392,A -90.000,B 90.000,C 0.000} C_DIS
LIN {X 97.766,Y -24.099,Z -177.830,A -90.000,B 90.000,C 0.000} C_DIS
LIN {X 97.733,Y -24.097,Z -178.175,A -90.000,B 90.000,C 0.000} C_DIS
LIN {X 97.492,Y -24.113,Z -180.365,A -90.000,B 90.000,C 0.000} C_DIS
LIN {X 97.469,Y -24.112,Z -180.601,A -90.000,B 90.000,C 0.000} C_DIS
LIN {X 97.441,Y -24.107,Z -180.883,A -90.000,B 90.000,C 0.000} C_DIS
LIN {X 97.423,Y -24.105,Z -181.061,A -90.000,B 90.000,C 0.000} C_DIS
LIN {X 97.244,Y -24.094,Z -182.671,A -90.000,B 90.000,C 0.000} C_DIS
LIN {X 97.196,Y -24.085,Z -183.150,A -90.000,B 90.000,C 0.000} C_DIS
LIN {X 97.135,Y -24.076,Z -183.787,A -90.000,B 90.000,C 0.000} C_DIS
LIN {X 97.025,Y -24.063,Z -184.834,A -90.000,B 90.000,C 0.000} C_DIS
LIN {X 96.955,Y -24.048,Z -185.579,A -90.000,B 90.000,C 0.000} C_DIS
LIN {X 96.838,Y -24.028,Z -186.808,A -90.000,B 90.000,C 0.000} C_DIS
LIN {X 96.692,Y -23.994,Z -188.444,A -90.000,B 90.000,C 0.000} C_DIS
LIN {X 96.483,Y -23.944,Z -190.910,A -90.000,B 90.000,C 0.000} C_DIS
LIN {X 96.454,Y -23.940,Z -191.174,A -90.000,B 90.000,C 0.000} C_DIS
LIN {X 96.188,Y -23.925,Z -193.449,A -90.000,B 90.000,C 0.000} C_DIS
LIN {X 96.167,Y -23.923,Z -193.607,A -90.000,B 90.000,C 0.000} C_DIS
LIN {X 96.099,Y -23.922,Z -194.062,A -90.000,B 90.000,C 0.000} C_DIS
LIN {X 95.870,Y -23.914,Z -195.570,A -90.000,B 90.000,C 0.000} C_DIS
LIN {X 95.689,Y -23.915,Z -196.715,A -90.000,B 90.000,C 0.000} C_DIS
LIN {X 95.634,Y -23.910,Z -197.023,A -90.000,B 90.000,C 0.000} C_DIS
LIN {X 95.197,Y -23.911,Z -199.221,A -90.000,B 90.000,C 0.000} C_DIS
LIN {X 94.979,Y -23.910,Z -200.314,A -90.000,B 90.000,C 0.000} C_DIS
LIN {X 94.930,Y -23.906,Z -200.542,A -90.000,B 90.000,C 0.000} C_DIS
LIN {X 94.221,Y -23.912,Z -203.541,A -90.000,B 90.000,C 0.000} C_DIS
LIN {X 93.928,Y -23.909,Z -204.796,A -90.000,B 90.000,C 0.000} C_DIS
LIN {X 93.502,Y -23.913,Z -206.471,A -90.000,B 90.000,C 0.000} C_DIS
LIN {X 93.190,Y -23.912,Z -207.684,A -90.000,B 90.000,C 0.000} C_DIS
LIN {X 92.697,Y -23.902,Z -209.619,A -90.000,B 90.000,C 0.000} C_DIS
LIN {X 92.016,Y -23.900,Z -212.189,A -90.000,B 90.000,C 0.000} C_DIS
LIN {X 91.307,Y -23.886,Z -214.901,A -90.000,B 90.000,C 0.000} C_DIS
LIN {X 90.761,Y -23.882,Z -216.959,A -90.000,B 90.000,C 0.000} C_DIS
LIN {X 89.848,Y -23.860,Z -220.439,A -90.000,B 90.000,C 0.000} C_DIS
LIN {X 89.504,Y -23.855,Z -221.768,A -90.000,B 90.000,C 0.000} C_DIS
LIN {X 89.126,Y -23.845,Z -223.240,A -90.000,B 90.000,C 0.000} C_DIS
LIN {X 88.639,Y -23.832,Z -225.144,A -90.000,B 90.000,C 0.000} C_DIS
LIN {X 88.473,Y -23.831,Z -225.795,A -90.000,B 90.000,C 0.000} C_DIS
LIN {X 88.240,Y -23.828,Z -226.657,A -90.000,B 90.000,C 0.000} C_DIS
LIN {X 87.542,Y -23.809,Z -229.265,A -90.000,B 90.000,C 0.000} C_DIS
LIN {X 86.995,Y -23.798,Z -231.319,A -90.000,B 90.000,C 0.000} C_DIS
LIN {X 86.899,Y -23.794,Z -231.651,A -90.000,B 90.000,C 0.000} C_DIS
LIN {X 86.610,Y -23.790,Z -232.626,A -90.000,B 90.000,C 0.000} C_DIS
LIN {X 86.151,Y -23.780,Z -234.181,A -90.000,B 90.000,C 0.000} C_DIS
LIN {X 85.644,Y -23.771,Z -235.912,A -90.000,B 90.000,C 0.000} C_DIS
LIN {X 85.300,Y -23.769,Z -237.077,A -90.000,B 90.000,C 0.000} C_DIS
LIN {X 85.190,Y -23.763,Z -237.422,A -90.000,B 90.000,C 0.000} C_DIS
LIN {X 84.366,Y -23.758,Z -239.862,A -90.000,B 90.000,C 0.000} C_DIS
LIN {X 83.130,Y -23.761,Z -243.561,A -90.000,B 90.000,C 0.000} C_DIS
LIN {X 83.130,Y -60.000,Z -243.561,A -90.000,B 90.000,C 0.000} C_DIS
LIN {X -105.589,Y -60.000,Z -243.561,A -90.000,B 90.000,C 0.000} C_DIS
LIN {X -105.589,Y -23.430,Z -243.561,A -90.000,B 90.000,C 0.000} C_DIS
LIN {X -105.371,Y -23.370,Z -243.403,A -90.000,B 90.000,C 0.000} C_DIS
LIN {X -105.130,Y -23.348,Z -243.236,A -90.000,B 90.000,C 0.000} C_DIS
LIN {X -102.580,Y -23.340,Z -241.515,A -90.000,B 90.000,C 0.000} C_DIS
LIN {X -94.679,Y -23.329,Z -236.295,A -90.000,B 90.000,C 0.000} C_DIS
LIN {X -86.510,Y -23.324,Z -231.030,A -90.000,B 90.000,C 0.000} C_DIS
LIN {X -78.042,Y -23.324,Z -225.736,A -90.000,B 90.000,C 0.000} C_DIS
LIN {X -73.816,Y -23.325,Z -223.191,A -90.000,B 90.000,C 0.000} C_DIS
LIN {X -70.213,Y -23.327,Z -221.022,A -90.000,B 90.000,C 0.000} C_DIS
LIN {X -69.390,Y -23.328,Z -220.529,A -90.000,B 90.000,C 0.000} C_DIS
LIN {X -68.818,Y -23.327,Z -220.190,A -90.000,B 90.000,C 0.000} C_DIS
LIN {X -62.174,Y -23.334,Z -216.287,A -90.000,B 90.000,C 0.000} C_DIS
LIN {X -59.639,Y -23.338,Z -214.812,A -90.000,B 90.000,C 0.000} C_DIS
LIN {X -52.889,Y -23.350,Z -210.903,A -90.000,B 90.000,C 0.000} C_DIS
LIN {X -52.146,Y -23.354,Z -210.465,A -90.000,B 90.000,C 0.000} C_DIS
LIN {X -47.265,Y -23.366,Z -207.643,A -90.000,B 90.000,C 0.000} C_DIS
LIN {X -45.751,Y -23.375,Z -206.768,A -90.000,B 90.000,C 0.000} C_DIS
LIN {X -42.186,Y -23.390,Z -204.669,A -90.000,B 90.000,C 0.000} C_DIS
LIN {X -42.153,Y -23.391,Z -204.649,A -90.000,B 90.000,C 0.000} C_DIS
LIN {X -40.288,Y -23.408,Z -203.522,A -90.000,B 90.000,C 0.000} C_DIS
LIN {X -38.808,Y -23.416,Z -202.625,A -90.000,B 90.000,C 0.000} C_DIS
LIN {X -37.045,Y -23.439,Z -201.517,A -90.000,B 90.000,C 0.000} C_DIS
LIN {X -35.775,Y -23.469,Z -200.687,A -90.000,B 90.000,C 0.000} C_DIS
LIN {X -35.599,Y -23.476,Z -200.568,A -90.000,B 90.000,C 0.000} C_DIS
LIN {X -34.436,Y -23.510,Z -199.765,A -90.000,B 90.000,C 0.000} C_DIS
LIN {X -33.027,Y -23.570,Z -198.763,A -90.000,B 90.000,C 0.000} C_DIS
LIN {X -32.220,Y -23.608,Z -198.193,A -90.000,B 90.000,C 0.000} C_DIS
LIN {X -31.726,Y -23.633,Z -197.845,A -90.000,B 90.000,C 0.000} C_DIS
LIN {X -31.004,Y -23.660,Z -197.318,A -90.000,B 90.000,C 0.000} C_DIS
LIN {X -29.057,Y -23.752,Z -195.874,A -90.000,B 90.000,C 0.000} C_DIS
LIN {X -28.581,Y -23.773,Z -195.516,A -90.000,B 90.000,C 0.000} C_DIS
LIN {X -26.519,Y -23.845,Z -193.912,A -90.000,B 90.000,C 0.000} C_DIS
LIN {X -25.973,Y -23.861,Z -193.482,A -90.000,B 90.000,C 0.000} C_DIS
LIN {X -25.487,Y -23.880,Z -193.093,A -90.000,B 90.000,C 0.000} C_DIS
LIN {X -25.243,Y -23.886,Z -192.889,A -90.000,B 90.000,C 0.000} C_DIS
LIN {X -23.732,Y -23.912,Z -191.609,A -90.000,B 90.000,C 0.000} C_DIS
LIN {X -23.103,Y -23.921,Z -191.080,A -90.000,B 90.000,C 0.000} C_DIS
LIN {X -22.843,Y -23.930,Z -190.854,A -90.000,B 90.000,C 0.000} C_DIS
LIN {X -21.581,Y -23.941,Z -189.690,A -90.000,B 90.000,C 0.000} C_DIS
LIN {X -20.935,Y -23.944,Z -189.092,A -90.000,B 90.000,C 0.000} C_DIS
LIN {X -20.475,Y -23.943,Z -188.670,A -90.000,B 90.000,C 0.000} C_DIS
LIN {X -20.359,Y -23.947,Z -188.558,A -90.000,B 90.000,C 0.000} C_DIS
LIN {X -19.558,Y -23.954,Z -187.754,A -90.000,B 90.000,C 0.000} C_DIS
LIN {X -18.029,Y -23.961,Z -186.210,A -90.000,B 90.000,C 0.000} C_DIS
LIN {X -17.872,Y -23.961,Z -186.053,A -90.000,B 90.000,C 0.000} C_DIS
LIN {X -17.654,Y -23.967,Z -185.825,A -90.000,B 90.000,C 0.000} C_DIS
LIN {X -17.267,Y -23.974,Z -185.406,A -90.000,B 90.000,C 0.000} C_DIS
LIN {X -16.193,Y -23.984,Z -184.222,A -90.000,B 90.000,C 0.000} C_DIS
LIN {X -15.327,Y -23.989,Z -183.261,A -90.000,B 90.000,C 0.000} C_DIS
LIN {X -15.174,Y -23.994,Z -183.086,A -90.000,B 90.000,C 0.000} C_DIS
LIN {X -13.998,Y -24.010,Z -181.649,A -90.000,B 90.000,C 0.000} C_DIS
LIN {X -12.940,Y -24.018,Z -180.341,A -90.000,B 90.000,C 0.000} C_DIS
LIN {X -12.688,Y -24.029,Z -180.017,A -90.000,B 90.000,C 0.000} C_DIS
LIN {X -12.301,Y -24.034,Z -179.487,A -90.000,B 90.000,C 0.000} C_DIS
LIN {X -11.932,Y -24.041,Z -178.978,A -90.000,B 90.000,C 0.000} C_DIS
LIN {X -10.676,Y -24.052,Z -177.205,A -90.000,B 90.000,C 0.000} C_DIS
LIN {X -10.462,Y -24.064,Z -176.887,A -90.000,B 90.000,C 0.000} C_DIS
LIN {X -9.979,Y -24.062,Z -176.088,A -90.000,B 90.000,C 0.000} C_DIS
LIN {X -9.177,Y -24.067,Z -174.743,A -90.000,B 90.000,C 0.000} C_DIS
LIN {X -8.762,Y -24.068,Z -174.044,A -90.000,B 90.000,C 0.000} C_DIS
LIN {X -8.593,Y -24.080,Z -173.740,A -90.000,B 90.000,C 0.000} C_DIS
LIN {X -7.903,Y -24.071,Z -172.318,A -90.000,B 90.000,C 0.000} C_DIS
LIN {X -7.692,Y -24.073,Z -171.875,A -90.000,B 90.000,C 0.000} C_DIS
LIN {X -7.239,Y -24.072,Z -170.914,A -90.000,B 90.000,C 0.000} C_DIS
LIN {X -7.110,Y -24.085,Z -170.615,A -90.000,B 90.000,C 0.000} C_DIS
LIN {X -6.667,Y -24.071,Z -169.365,A -90.000,B 90.000,C 0.000} C_DIS
LIN {X -6.515,Y -24.064,Z -168.934,A -90.000,B 90.000,C 0.000} C_DIS
LIN {X -6.123,Y -24.061,Z -167.785,A -90.000,B 90.000,C 0.000} C_DIS
LIN {X -6.058,Y -24.072,Z -167.562,A -90.000,B 90.000,C 0.000} C_DIS
LIN {X -5.662,Y -24.033,Z -165.561,A -90.000,B 90.000,C 0.000} C_DIS
LIN {X -5.565,Y -24.030,Z -165.045,A -90.000,B 90.000,C 0.000} C_DIS
LIN {X -5.563,Y -24.026,Z -164.997,A -90.000,B 90.000,C 0.000} C_DIS
LIN {X -5.548,Y -23.997,Z -163.121,A -90.000,B 90.000,C 0.000} C_DIS
LIN {X -5.575,Y -23.970,Z -162.955,A -90.000,B 90.000,C 0.000} C_DIS
LIN {X -5.866,Y -23.946,Z -161.951,A -90.000,B 90.000,C 0.000} C_DIS
LIN {X -5.890,Y -23.936,Z -161.898,A -90.000,B 90.000,C 0.000} C_DIS
LIN {X -6.071,Y -23.858,Z -161.487,A -90.000,B 90.000,C 0.000} C_DIS
LIN {X -6.337,Y -23.849,Z -161.045,A -90.000,B 90.000,C 0.000} C_DIS
LIN {X -6.646,Y -23.779,Z -160.638,A -90.000,B 90.000,C 0.000} C_DIS
LIN {X -6.724,Y -23.764,Z -160.531,A -90.000,B 90.000,C 0.000} C_DIS
LIN {X -6.814,Y -23.742,Z -160.397,A -90.000,B 90.000,C 0.000} C_DIS
LIN {X -7.183,Y -23.739,Z -160.004,A -90.000,B 90.000,C 0.000} C_DIS
LIN {X -7.363,Y -23.718,Z -159.834,A -90.000,B 90.000,C 0.000} C_DIS
LIN {X -7.449,Y -23.711,Z -159.750,A -90.000,B 90.000,C 0.000} C_DIS
LIN {X -7.765,Y -23.672,Z -159.421,A -90.000,B 90.000,C 0.000} C_DIS
LIN {X -8.291,Y -23.670,Z -158.986,A -90.000,B 90.000,C 0.000} C_DIS
LIN {X -8.552,Y -23.661,Z -158.756,A -90.000,B 90.000,C 0.000} C_DIS
LIN {X -9.244,Y -23.623,Z -158.157,A -90.000,B 90.000,C 0.000} C_DIS
LIN {X -10.180,Y -23.602,Z -157.397,A -90.000,B 90.000,C 0.000} C_DIS
LIN {X -10.498,Y -23.597,Z -157.132,A -90.000,B 90.000,C 0.000} C_DIS
LIN {X -11.247,Y -23.583,Z -156.537,A -90.000,B 90.000,C 0.000} C_DIS
LIN {X -12.308,Y -23.553,Z -155.669,A -90.000,B 90.000,C 0.000} C_DIS
LIN {X -12.673,Y -23.549,Z -155.362,A -90.000,B 90.000,C 0.000} C_DIS
LIN {X -13.026,Y -23.548,Z -155.073,A -90.000,B 90.000,C 0.000} C_DIS
LIN {X -14.501,Y -23.518,Z -153.875,A -90.000,B 90.000,C 0.000} C_DIS
LIN {X -14.935,Y -23.516,Z -153.511,A -90.000,B 90.000,C 0.000} C_DIS
LIN {X -15.249,Y -23.516,Z -153.252,A -90.000,B 90.000,C 0.000} C_DIS
LIN {X -17.053,Y -23.494,Z -151.771,A -90.000,B 90.000,C 0.000} C_DIS
LIN {X -17.361,Y -23.494,Z -151.511,A -90.000,B 90.000,C 0.000} C_DIS
LIN {X -17.874,Y -23.493,Z -151.076,A -90.000,B 90.000,C 0.000} C_DIS
LIN {X -20.278,Y -23.485,Z -149.060,A -90.000,B 90.000,C 0.000} C_DIS
LIN {X -20.464,Y -23.481,Z -148.894,A -90.000,B 90.000,C 0.000} C_DIS
LIN {X -23.520,Y -23.481,Z -146.132,A -90.000,B 90.000,C 0.000} C_DIS
LIN {X -23.725,Y -23.475,Z -145.926,A -90.000,B 90.000,C 0.000} C_DIS
LIN {X -26.415,Y -23.468,Z -143.175,A -90.000,B 90.000,C 0.000} C_DIS
LIN {X -26.844,Y -23.466,Z -142.734,A -90.000,B 90.000,C 0.000} C_DIS
LIN {X -27.084,Y -23.465,Z -142.484,A -90.000,B 90.000,C 0.000} C_DIS
LIN {X -27.261,Y -23.457,Z -142.272,A -90.000,B 90.000,C 0.000} C_DIS
LIN {X -28.177,Y -23.453,Z -141.150,A -90.000,B 90.000,C 0.000} C_DIS
LIN {X -28.990,Y -23.436,Z -140.162,A -90.000,B 90.000,C 0.000} C_DIS
LIN {X -29.740,Y -23.418,Z -139.247,A -90.000,B 90.000,C 0.000} C_DIS
LIN {X -30.093,Y -23.400,Z -138.820,A -90.000,B 90.000,C 0.000} C_DIS
LIN {X -30.355,Y -23.386,Z -138.491,A -90.000,B 90.000,C 0.000} C_DIS
LIN {X -30.576,Y -23.365,Z -138.154,A -90.000,B 90.000,C 0.000} C_DIS
LIN {X -30.852,Y -23.350,Z -137.724,A -90.000,B 90.000,C 0.000} C_DIS
LIN {X -31.419,Y -23.329,Z -136.836,A -90.000,B 90.000,C 0.000} C_DIS
LIN {X -31.807,Y -23.319,Z -136.224,A -90.000,B 90.000,C 0.000} C_DIS
LIN {X -32.431,Y -23.310,Z -135.270,A -90.000,B 90.000,C 0.000} C_DIS
LIN {X -32.887,Y -23.308,Z -134.570,A -90.000,B 90.000,C 0.000} C_DIS
LIN {X -32.887,Y -60.000,Z -134.570,A -90.000,B 90.000,C 0.000} C_DIS
LIN {X -38.830,Y -60.000,Z -124.589,A -90.000,B 90.000,C 0.000} C_DIS
LIN {X -38.830,Y -23.308,Z -124.589,A -90.000,B 90.000,C 0.000} C_DIS
LIN {X -39.763,Y -23.309,Z -122.731,A -90.000,B 90.000,C 0.000} C_DIS
LIN {X -40.430,Y -23.310,Z -121.314,A -90.000,B 90.000,C 0.000} C_DIS
LIN {X -40.748,Y -23.310,Z -120.596,A -90.000,B 90.000,C 0.000} C_DIS
LIN {X -40.984,Y -23.312,Z -120.125,A -90.000,B 90.000,C 0.000} C_DIS
LIN {X -41.007,Y -23.313,Z -120.078,A -90.000,B 90.000,C 0.000} C_DIS
LIN {X -41.493,Y -23.323,Z -119.102,A -90.000,B 90.000,C 0.000} C_DIS
LIN {X -41.675,Y -23.324,Z -118.675,A -90.000,B 90.000,C 0.000} C_DIS
LIN {X -42.022,Y -23.337,Z -118.039,A -90.000,B 90.000,C 0.000} C_DIS
LIN {X -42.302,Y -23.355,Z -117.522,A -90.000,B 90.000,C 0.000} C_DIS
LIN {X -42.492,Y -23.361,Z -117.174,A -90.000,B 90.000,C 0.000} C_DIS
LIN {X -42.563,Y -23.361,Z -117.025,A -90.000,B 90.000,C 0.000} C_DIS
LIN {X -43.012,Y -23.389,Z -116.301,A -90.000,B 90.000,C 0.000} C_DIS
LIN {X -43.239,Y -23.408,Z -115.933,A -90.000,B 90.000,C 0.000} C_DIS
LIN {X -43.668,Y -23.421,Z -115.244,A -90.000,B 90.000,C 0.000} C_DIS
LIN {X -43.700,Y -23.421,Z -115.188,A -90.000,B 90.000,C 0.000} C_DIS
LIN {X -44.179,Y -23.450,Z -114.489,A -90.000,B 90.000,C 0.000} C_DIS
LIN {X -44.366,Y -23.464,Z -114.215,A -90.000,B 90.000,C 0.000} C_DIS
LIN {X -45.179,Y -23.479,Z -113.047,A -90.000,B 90.000,C 0.000} C_DIS
LIN {X -45.371,Y -23.481,Z -112.763,A -90.000,B 90.000,C 0.000} C_DIS
LIN {X -45.964,Y -23.500,Z -111.944,A -90.000,B 90.000,C 0.000} C_DIS
LIN {X -46.992,Y -23.510,Z -110.540,A -90.000,B 90.000,C 0.000} C_DIS
LIN {X -47.641,Y -23.510,Z -109.662,A -90.000,B 90.000,C 0.000} C_DIS
LIN {X -48.301,Y -23.514,Z -108.780,A -90.000,B 90.000,C 0.000} C_DIS
LIN {X -49.103,Y -23.513,Z -107.739,A -90.000,B 90.000,C 0.000} C_DIS
LIN {X -49.532,Y -23.516,Z -107.178,A -90.000,B 90.000,C 0.000} C_DIS
LIN {X -50.003,Y -23.517,Z -106.549,A -90.000,B 90.000,C 0.000} C_DIS
LIN {X -50.119,Y -23.515,Z -106.400,A -90.000,B 90.000,C 0.000} C_DIS
LIN {X -50.402,Y -23.512,Z -106.028,A -90.000,B 90.000,C 0.000} C_DIS
LIN {X -51.518,Y -23.508,Z -104.547,A -90.000,B 90.000,C 0.000} C_DIS
LIN {X -51.688,Y -23.510,Z -104.328,A -90.000,B 90.000,C 0.000} C_DIS
LIN {X -52.383,Y -23.506,Z -103.448,A -90.000,B 90.000,C 0.000} C_DIS
LIN {X -52.655,Y -23.503,Z -103.098,A -90.000,B 90.000,C 0.000} C_DIS
LIN {X -52.782,Y -23.500,Z -102.927,A -90.000,B 90.000,C 0.000} C_DIS
LIN {X -53.337,Y -23.493,Z -102.181,A -90.000,B 90.000,C 0.000} C_DIS
LIN {X -54.789,Y -23.495,Z -100.290,A -90.000,B 90.000,C 0.000} C_DIS
LIN {X -54.992,Y -23.493,Z -100.018,A -90.000,B 90.000,C 0.000} C_DIS
LIN {X -55.128,Y -23.494,Z -99.841,A -90.000,B 90.000,C 0.000} C_DIS
LIN {X -55.692,Y -23.493,Z -99.079,A -90.000,B 90.000,C 0.000} C_DIS
LIN {X -56.647,Y -23.494,Z -97.785,A -90.000,B 90.000,C 0.000} C_DIS
LIN {X -56.912,Y -23.497,Z -97.437,A -90.000,B 90.000,C 0.000} C_DIS
LIN {X -57.513,Y -23.497,Z -96.652,A -90.000,B 90.000,C 0.000} C_DIS
LIN {X -58.267,Y -23.497,Z -95.640,A -90.000,B 90.000,C 0.000} C_DIS
LIN {X -59.551,Y -23.499,Z -93.971,A -90.000,B 90.000,C 0.000} C_DIS
LIN {X -60.019,Y -23.502,Z -93.371,A -90.000,B 90.000,C 0.000} C_DIS
LIN {X -60.267,Y -23.501,Z -93.051,A -90.000,B 90.000,C 0.000} C_DIS
LIN {X -60.714,Y -23.498,Z -92.466,A -90.000,B 90.000,C 0.000} C_DIS
LIN {X -61.242,Y -23.500,Z -91.769,A -90.000,B 90.000,C 0.000} C_DIS
LIN {X -61.550,Y -23.505,Z -91.376,A -90.000,B 90.000,C 0.000} C_DIS
LIN {X -61.848,Y -23.510,Z -91.014,A -90.000,B 90.000,C 0.000} C_DIS
LIN {X -62.260,Y -23.510,Z -90.519,A -90.000,B 90.000,C 0.000} C_DIS
LIN {X -63.465,Y -23.509,Z -89.033,A -90.000,B 90.000,C 0.000} C_DIS
LIN {X -63.750,Y -23.516,Z -88.705,A -90.000,B 90.000,C 0.000} C_DIS
LIN {X -64.849,Y -23.513,Z -87.456,A -90.000,B 90.000,C 0.000} C_DIS
LIN {X -65.295,Y -23.510,Z -86.936,A -90.000,B 90.000,C 0.000} C_DIS
LIN {X -65.583,Y -23.516,Z -86.619,A -90.000,B 90.000,C 0.000} C_DIS
LIN {X -66.546,Y -23.513,Z -85.573,A -90.000,B 90.000,C 0.000} C_DIS
LIN {X -67.066,Y -23.509,Z -84.998,A -90.000,B 90.000,C 0.000} C_DIS
LIN {X -67.358,Y -23.514,Z -84.685,A -90.000,B 90.000,C 0.000} C_DIS
LIN {X -68.301,Y -23.516,Z -83.665,A -90.000,B 90.000,C 0.000} C_DIS
LIN {X -68.813,Y -23.518,Z -83.110,A -90.000,B 90.000,C 0.000} C_DIS
LIN {X -69.353,Y -23.522,Z -82.538,A -90.000,B 90.000,C 0.000} C_DIS
LIN {X -69.911,Y -23.524,Z -81.949,A -90.000,B 90.000,C 0.000} C_DIS
LIN {X -70.508,Y -23.524,Z -81.309,A -90.000,B 90.000,C 0.000} C_DIS
LIN {X -70.807,Y -23.529,Z -80.998,A -90.000,B 90.000,C 0.000} C_DIS
LIN {X -71.473,Y -23.535,Z -80.310,A -90.000,B 90.000,C 0.000} C_DIS
LIN {X -71.784,Y -23.538,Z -79.983,A -90.000,B 90.000,C 0.000} C_DIS
LIN {X -72.046,Y -23.539,Z -79.704,A -90.000,B 90.000,C 0.000} C_DIS
LIN {X -72.496,Y -23.548,Z -79.244,A -90.000,B 90.000,C 0.000} C_DIS
LIN {X -72.721,Y -23.551,Z -79.015,A -90.000,B 90.000,C 0.000} C_DIS
LIN {X -73.480,Y -23.566,Z -78.239,A -90.000,B 90.000,C 0.000} C_DIS
LIN {X -73.882,Y -23.585,Z -77.855,A -90.000,B 90.000,C 0.000} C_DIS
LIN {X -74.636,Y -23.601,Z -77.160,A -90.000,B 90.000,C 0.000} C_DIS
LIN {X -74.701,Y -23.605,Z -77.106,A -90.000,B 90.000,C 0.000} C_DIS
LIN {X -75.011,Y -23.636,Z -76.870,A -90.000,B 90.000,C 0.000} C_DIS
LIN {X -75.057,Y -23.638,Z -76.836,A -90.000,B 90.000,C 0.000} C_DIS
LIN {X -75.112,Y -23.654,Z -76.822,A -90.000,B 90.000,C 0.000} C_DIS
LIN {X -75.355,Y -23.723,Z -76.748,A -90.000,B 90.000,C 0.000} C_DIS
LIN {X -75.417,Y -23.742,Z -76.730,A -90.000,B 90.000,C 0.000} C_DIS
LIN {X -75.902,Y -23.730,Z -76.691,A -90.000,B 90.000,C 0.000} C_DIS
LIN {X -75.951,Y -23.731,Z -76.686,A -90.000,B 90.000,C 0.000} C_DIS
LIN {X -76.167,Y -23.743,Z -76.676,A -90.000,B 90.000,C 0.000} C_DIS
LIN {X -76.525,Y -23.749,Z -76.667,A -90.000,B 90.000,C 0.000} C_DIS
LIN {X -76.976,Y -23.733,Z -76.625,A -90.000,B 90.000,C 0.000} C_DIS
LIN {X -77.044,Y -23.730,Z -76.615,A -90.000,B 90.000,C 0.000} C_DIS
LIN {X -77.148,Y -23.732,Z -76.600,A -90.000,B 90.000,C 0.000} C_DIS
LIN {X -77.507,Y -23.722,Z -76.526,A -90.000,B 90.000,C 0.000} C_DIS
LIN {X -77.595,Y -23.722,Z -76.507,A -90.000,B 90.000,C 0.000} C_DIS
LIN {X -77.828,Y -23.724,Z -76.453,A -90.000,B 90.000,C 0.000} C_DIS
LIN {X -78.229,Y -23.721,Z -76.350,A -90.000,B 90.000,C 0.000} C_DIS
LIN {X -78.551,Y -23.712,Z -76.268,A -90.000,B 90.000,C 0.000} C_DIS
LIN {X -78.750,Y -23.705,Z -76.213,A -90.000,B 90.000,C 0.000} C_DIS
LIN {X -79.235,Y -23.690,Z -76.051,A -90.000,B 90.000,C 0.000} C_DIS
LIN {X -79.617,Y -23.683,Z -75.917,A -90.000,B 90.000,C 0.000} C_DIS
LIN {X -80.270,Y -23.690,Z -75.653,A -90.000,B 90.000,C 0.000} C_DIS
LIN {X -80.486,Y -23.681,Z -75.545,A -90.000,B 90.000,C 0.000} C_DIS
LIN {X -80.687,Y -23.678,Z -75.441,A -90.000,B 90.000,C 0.000} C_DIS
LIN {X -80.940,Y -23.665,Z -75.296,A -90.000,B 90.000,C 0.000} C_DIS
LIN {X -81.249,Y -23.657,Z -75.115,A -90.000,B 90.000,C 0.000} C_DIS
LIN {X -81.839,Y -23.648,Z -74.763,A -90.000,B 90.000,C 0.000} C_DIS
LIN {X -82.172,Y -23.634,Z -74.548,A -90.000,B 90.000,C 0.000} C_DIS
LIN {X -82.352,Y -23.630,Z -74.424,A -90.000,B 90.000,C 0.000} C_DIS
LIN {X -82.642,Y -23.629,Z -74.215,A -90.000,B 90.000,C 0.000} C_DIS
LIN {X -82.836,Y -23.623,Z -74.061,A -90.000,B 90.000,C 0.000} C_DIS
LIN {X -83.200,Y -23.623,Z -73.763,A -90.000,B 90.000,C 0.000} C_DIS
LIN {X -83.493,Y -23.623,Z -73.515,A -90.000,B 90.000,C 0.000} C_DIS
LIN {X -83.554,Y -23.624,Z -73.462,A -90.000,B 90.000,C 0.000} C_DIS
LIN {X -83.933,Y -23.630,Z -73.081,A -90.000,B 90.000,C 0.000} C_DIS
LIN {X -84.245,Y -23.638,Z -72.764,A -90.000,B 90.000,C 0.000} C_DIS
LIN {X -84.496,Y -23.637,Z -72.499,A -90.000,B 90.000,C 0.000} C_DIS
LIN {X -84.614,Y -23.642,Z -72.369,A -90.000,B 90.000,C 0.000} C_DIS
LIN {X -84.817,Y -23.651,Z -72.129,A -90.000,B 90.000,C 0.000} C_DIS
LIN {X -84.915,Y -23.653,Z -72.000,A -90.000,B 90.000,C 0.000} C_DIS
LIN {X -85.118,Y -23.660,Z -71.725,A -90.000,B 90.000,C 0.000} C_DIS
LIN {X -85.396,Y -23.679,Z -71.326,A -90.000,B 90.000,C 0.000} C_DIS
LIN {X -85.650,Y -23.701,Z -70.968,A -90.000,B 90.000,C 0.000} C_DIS
LIN {X -85.716,Y -23.708,Z -70.856,A -90.000,B 90.000,C 0.000} C_DIS
LIN {X -85.787,Y -23.718,Z -70.734,A -90.000,B 90.000,C 0.000} C_DIS
LIN {X -85.971,Y -23.750,Z -70.430,A -90.000,B 90.000,C 0.000} C_DIS
LIN {X -86.059,Y -23.770,Z -70.278,A -90.000,B 90.000,C 0.000} C_DIS
LIN {X -86.314,Y -23.835,Z -69.891,A -90.000,B 90.000,C 0.000} C_DIS
LIN {X -86.396,Y -23.862,Z -69.757,A -90.000,B 90.000,C 0.000} C_DIS
LIN {X -86.491,Y -23.901,Z -69.591,A -90.000,B 90.000,C 0.000} C_DIS
LIN {X -86.705,Y -23.993,Z -69.228,A -90.000,B 90.000,C 0.000} C_DIS
LIN {X -86.890,Y -24.090,Z -68.852,A -90.000,B 90.000,C 0.000} C_DIS
LIN {X -87.009,Y -24.154,Z -68.607,A -90.000,B 90.000,C 0.000} C_DIS
LIN {X -87.049,Y -24.179,Z -68.517,A -90.000,B 90.000,C 0.000} C_DIS
LIN {X -87.174,Y -24.266,Z -68.219,A -90.000,B 90.000,C 0.000} C_DIS
LIN {X -87.225,Y -24.305,Z -68.097,A -90.000,B 90.000,C 0.000} C_DIS
LIN {X -87.259,Y -24.309,Z -68.056,A -90.000,B 90.000,C 0.000} C_DIS
LIN {X -87.332,Y -24.320,Z -67.962,A -90.000,B 90.000,C 0.000} C_DIS
LIN {X -87.565,Y -24.334,Z -67.703,A -90.000,B 90.000,C 0.000} C_DIS
LIN {X -87.725,Y -24.339,Z -67.544,A -90.000,B 90.000,C 0.000} C_DIS
LIN {X -87.892,Y -24.336,Z -67.396,A -90.000,B 90.000,C 0.000} C_DIS
LIN {X -88.125,Y -24.320,Z -67.214,A -90.000,B 90.000,C 0.000} C_DIS
LIN {X -88.422,Y -24.309,Z -66.980,A -90.000,B 90.000,C 0.000} C_DIS
LIN {X -88.638,Y -24.295,Z -66.822,A -90.000,B 90.000,C 0.000} C_DIS
LIN {X -88.726,Y -24.292,Z -66.760,A -90.000,B 90.000,C 0.000} C_DIS
LIN {X -89.095,Y -24.283,Z -66.491,A -90.000,B 90.000,C 0.000} C_DIS
LIN {X -89.216,Y -24.278,Z -66.405,A -90.000,B 90.000,C 0.000} C_DIS
LIN {X -90.024,Y -24.271,Z -65.849,A -90.000,B 90.000,C 0.000} C_DIS
LIN {X -90.354,Y -24.272,Z -65.617,A -90.000,B 90.000,C 0.000} C_DIS
LIN {X -90.679,Y -24.272,Z -65.394,A -90.000,B 90.000,C 0.000} C_DIS
LIN {X -91.096,Y -24.268,Z -65.104,A -90.000,B 90.000,C 0.000} C_DIS
LIN {X -91.369,Y -24.269,Z -64.904,A -90.000,B 90.000,C 0.000} C_DIS
LIN {X -92.146,Y -24.266,Z -64.343,A -90.000,B 90.000,C 0.000} C_DIS
LIN {X -92.437,Y -24.267,Z -64.117,A -90.000,B 90.000,C 0.000} C_DIS
LIN {X -93.066,Y -24.276,Z -63.617,A -90.000,B 90.000,C 0.000} C_DIS
LIN {X -93.207,Y -24.276,Z -63.502,A -90.000,B 90.000,C 0.000} C_DIS
LIN {X -93.361,Y -24.279,Z -63.369,A -90.000,B 90.000,C 0.000} C_DIS
LIN {X -93.684,Y -24.280,Z -63.087,A -90.000,B 90.000,C 0.000} C_DIS
LIN {X -93.758,Y -24.282,Z -63.019,A -90.000,B 90.000,C 0.000} C_DIS
LIN {X -94.187,Y -24.302,Z -62.614,A -90.000,B 90.000,C 0.000} C_DIS
LIN {X -94.601,Y -24.301,Z -62.196,A -90.000,B 90.000,C 0.000} C_DIS
LIN {X -94.698,Y -24.304,Z -62.092,A -90.000,B 90.000,C 0.000} C_DIS
LIN {X -94.995,Y -24.320,Z -61.756,A -90.000,B 90.000,C 0.000} C_DIS
LIN {X -95.441,Y -24.331,Z -61.248,A -90.000,B 90.000,C 0.000} C_DIS
LIN {X -95.664,Y -24.339,Z -60.985,A -90.000,B 90.000,C 0.000} C_DIS
LIN {X -95.781,Y -24.347,Z -60.840,A -90.000,B 90.000,C 0.000} C_DIS
LIN {X -96.118,Y -24.380,Z -60.386,A -90.000,B 90.000,C 0.000} C_DIS
LIN {X -96.299,Y -24.400,Z -60.144,A -90.000,B 90.000,C 0.000} C_DIS
LIN {X -96.364,Y -24.410,Z -60.052,A -90.000,B 90.000,C 0.000} C_DIS
LIN {X -96.484,Y -24.431,Z -59.876,A -90.000,B 90.000,C 0.000} C_DIS
LIN {X -96.554,Y -24.438,Z -59.763,A -90.000,B 90.000,C 0.000} C_DIS
LIN {X -96.719,Y -24.457,Z -59.491,A -90.000,B 90.000,C 0.000} C_DIS
LIN {X -96.955,Y -24.470,Z -59.142,A -90.000,B 90.000,C 0.000} C_DIS
LIN {X -97.147,Y -24.485,Z -58.844,A -90.000,B 90.000,C 0.000} C_DIS
LIN {X -97.491,Y -24.529,Z -58.247,A -90.000,B 90.000,C 0.000} C_DIS
LIN {X -97.763,Y -24.543,Z -57.752,A -90.000,B 90.000,C 0.000} C_DIS
LIN {X -97.820,Y -24.548,Z -57.633,A -90.000,B 90.000,C 0.000} C_DIS
LIN {X -98.019,Y -24.572,Z -57.189,A -90.000,B 90.000,C 0.000} C_DIS
LIN {X -98.082,Y -24.575,Z -57.038,A -90.000,B 90.000,C 0.000} C_DIS
LIN {X -98.117,Y -24.579,Z -56.946,A -90.000,B 90.000,C 0.000} C_DIS
LIN {X -98.219,Y -24.593,Z -56.647,A -90.000,B 90.000,C 0.000} C_DIS
LIN {X -98.253,Y -24.600,Z -56.531,A -90.000,B 90.000,C 0.000} C_DIS
LIN {X -98.320,Y -24.622,Z -56.240,A -90.000,B 90.000,C 0.000} C_DIS
LIN {X -98.336,Y -24.627,Z -56.168,A -90.000,B 90.000,C 0.000} C_DIS
LIN {X -98.361,Y -24.636,Z -56.025,A -90.000,B 90.000,C 0.000} C_DIS
LIN {X -98.397,Y -24.649,Z -55.772,A -90.000,B 90.000,C 0.000} C_DIS
LIN {X -98.412,Y -24.667,Z -55.522,A -90.000,B 90.000,C 0.000} C_DIS
LIN {X -98.407,Y -24.686,Z -55.357,A -90.000,B 90.000,C 0.000} C_DIS
LIN {X -98.399,Y -24.695,Z -55.233,A -90.000,B 90.000,C 0.000} C_DIS
LIN {X -98.555,Y -24.645,Z -55.033,A -90.000,B 90.000,C 0.000} C_DIS
LIN {X -98.736,Y -24.577,Z -54.792,A -90.000,B 90.000,C 0.000} C_DIS
LIN {X -98.795,Y -24.554,Z -54.707,A -90.000,B 90.000,C 0.000} C_DIS
LIN {X -98.873,Y -24.523,Z -54.589,A -90.000,B 90.000,C 0.000} C_DIS
LIN {X -98.968,Y -24.478,Z -54.439,A -90.000,B 90.000,C 0.000} C_DIS
LIN {X -99.102,Y -24.406,Z -54.210,A -90.000,B 90.000,C 0.000} C_DIS
LIN {X -99.240,Y -24.319,Z -53.957,A -90.000,B 90.000,C 0.000} C_DIS
LIN {X -99.327,Y -24.263,Z -53.790,A -90.000,B 90.000,C 0.000} C_DIS
LIN {X -99.418,Y -24.200,Z -53.607,A -90.000,B 90.000,C 0.000} C_DIS
LIN {X -99.567,Y -24.094,Z -53.292,A -90.000,B 90.000,C 0.000} C_DIS
LIN {X -99.623,Y -24.044,Z -53.156,A -90.000,B 90.000,C 0.000} C_DIS
LIN {X -99.703,Y -23.965,Z -52.925,A -90.000,B 90.000,C 0.000} C_DIS
LIN {X -99.729,Y -23.937,Z -52.843,A -90.000,B 90.000,C 0.000} C_DIS
LIN {X -99.744,Y -23.918,Z -52.792,A -90.000,B 90.000,C 0.000} C_DIS
LIN {X -99.867,Y -23.931,Z -52.631,A -90.000,B 90.000,C 0.000} C_DIS
LIN {X -100.011,Y -23.949,Z -52.443,A -90.000,B 90.000,C 0.000} C_DIS
LIN {X -100.212,Y -23.980,Z -52.159,A -90.000,B 90.000,C 0.000} C_DIS
LIN {X -100.485,Y -24.032,Z -51.734,A -90.000,B 90.000,C 0.000} C_DIS
LIN {X -100.718,Y -24.075,Z -51.354,A -90.000,B 90.000,C 0.000} C_DIS
LIN {X -100.777,Y -24.085,Z -51.257,A -90.000,B 90.000,C 0.000} C_DIS
LIN {X -100.924,Y -24.118,Z -51.001,A -90.000,B 90.000,C 0.000} C_DIS
LIN {X -101.061,Y -24.146,Z -50.732,A -90.000,B 90.000,C 0.000} C_DIS
LIN {X -101.136,Y -24.166,Z -50.575,A -90.000,B 90.000,C 0.000} C_DIS
LIN {X -101.237,Y -24.190,Z -50.340,A -90.000,B 90.000,C 0.000} C_DIS
LIN {X -101.351,Y -24.222,Z -50.055,A -90.000,B 90.000,C 0.000} C_DIS
LIN {X -101.434,Y -24.246,Z -49.836,A -90.000,B 90.000,C 0.000} C_DIS
LIN {X -101.486,Y -24.263,Z -49.691,A -90.000,B 90.000,C 0.000} C_DIS
LIN {X -101.565,Y -24.280,Z -49.436,A -90.000,B 90.000,C 0.000} C_DIS
LIN {X -101.633,Y -24.298,Z -49.190,A -90.000,B 90.000,C 0.000} C_DIS
LIN {X -101.687,Y -24.312,Z -48.987,A -90.000,B 90.000,C 0.000} C_DIS
LIN {X -101.696,Y -24.316,Z -48.948,A -90.000,B 90.000,C 0.000} C_DIS
LIN {X -101.721,Y -24.330,Z -48.823,A -90.000,B 90.000,C 0.000} C_DIS
LIN {X -101.761,Y -24.369,Z -48.539,A -90.000,B 90.000,C 0.000} C_DIS
LIN {X -101.800,Y -24.398,Z -48.167,A -90.000,B 90.000,C 0.000} C_DIS
LIN {X -101.816,Y -24.410,Z -47.985,A -90.000,B 90.000,C 0.000} C_DIS
LIN {X -101.820,Y -24.423,Z -47.852,A -90.000,B 90.000,C 0.000} C_DIS
LIN {X -101.817,Y -24.444,Z -47.570,A -90.000,B 90.000,C 0.000} C_DIS
LIN {X -101.813,Y -24.450,Z -47.431,A -90.000,B 90.000,C 0.000} C_DIS
LIN {X -101.809,Y -24.456,Z -47.334,A -90.000,B 90.000,C 0.000} C_DIS
LIN {X -101.803,Y -24.461,Z -47.272,A -90.000,B 90.000,C 0.000} C_DIS
LIN {X -101.776,Y -24.480,Z -47.064,A -90.000,B 90.000,C 0.000} C_DIS
LIN {X -101.756,Y -24.492,Z -46.931,A -90.000,B 90.000,C 0.000} C_DIS
LIN {X -101.724,Y -24.500,Z -46.750,A -90.000,B 90.000,C 0.000} C_DIS
LIN {X -101.700,Y -24.506,Z -46.629,A -90.000,B 90.000,C 0.000} C_DIS
LIN {X -101.656,Y -24.509,Z -46.426,A -90.000,B 90.000,C 0.000} C_DIS
LIN {X -101.617,Y -24.515,Z -46.290,A -90.000,B 90.000,C 0.000} C_DIS
LIN {X -101.573,Y -24.521,Z -46.167,A -90.000,B 90.000,C 0.000} C_DIS
LIN {X -101.507,Y -24.531,Z -45.999,A -90.000,B 90.000,C 0.000} C_DIS
LIN {X -101.454,Y -24.530,Z -45.872,A -90.000,B 90.000,C 0.000} C_DIS
LIN {X -101.270,Y -24.536,Z -45.481,A -90.000,B 90.000,C 0.000} C_DIS
LIN {X -101.223,Y -24.539,Z -45.389,A -90.000,B 90.000,C 0.000} C_DIS
LIN {X -101.143,Y -24.538,Z -45.261,A -90.000,B 90.000,C 0.000} C_DIS
LIN {X -101.052,Y -24.539,Z -45.119,A -90.000,B 90.000,C 0.000} C_DIS
LIN {X -100.950,Y -24.536,Z -44.969,A -90.000,B 90.000,C 0.000} C_DIS
LIN {X -100.832,Y -24.540,Z -44.819,A -90.000,B 90.000,C 0.000} C_DIS
LIN {X -100.631,Y -24.536,Z -44.573,A -90.000,B 90.000,C 0.000} C_DIS
LIN {X -100.376,Y -24.527,Z -44.301,A -90.000,B 90.000,C 0.000} C_DIS
LIN {X -100.308,Y -24.525,Z -44.234,A -90.000,B 90.000,C 0.000} C_DIS
LIN {X -100.195,Y -24.523,Z -44.135,A -90.000,B 90.000,C 0.000} C_DIS
LIN {X -100.121,Y -24.523,Z -44.074,A -90.000,B 90.000,C 0.000} C_DIS
LIN {X -99.987,Y -24.513,Z -43.969,A -90.000,B 90.000,C 0.000} C_DIS
LIN {X -99.891,Y -24.504,Z -43.888,A -90.000,B 90.000,C 0.000} C_DIS
LIN {X -99.781,Y -24.498,Z -43.805,A -90.000,B 90.000,C 0.000} C_DIS
LIN {X -99.533,Y -24.486,Z -43.626,A -90.000,B 90.000,C 0.000} C_DIS
LIN {X -99.412,Y -24.472,Z -43.547,A -90.000,B 90.000,C 0.000} C_DIS
LIN {X -99.234,Y -24.458,Z -43.444,A -90.000,B 90.000,C 0.000} C_DIS
LIN {X -99.051,Y -24.441,Z -43.343,A -90.000,B 90.000,C 0.000} C_DIS
LIN {X -98.923,Y -24.431,Z -43.279,A -90.000,B 90.000,C 0.000} C_DIS
LIN {X -98.745,Y -24.419,Z -43.196,A -90.000,B 90.000,C 0.000} C_DIS
LIN {X -98.473,Y -24.388,Z -43.068,A -90.000,B 90.000,C 0.000} C_DIS
LIN {X -98.348,Y -24.376,Z -43.019,A -90.000,B 90.000,C 0.000} C_DIS
LIN {X -98.189,Y -24.363,Z -42.963,A -90.000,B 90.000,C 0.000} C_DIS
LIN {X -98.040,Y -24.339,Z -42.916,A -90.000,B 90.000,C 0.000} C_DIS
LIN {X -97.949,Y -24.326,Z -42.890,A -90.000,B 90.000,C 0.000} C_DIS
LIN {X -97.817,Y -24.312,Z -42.860,A -90.000,B 90.000,C 0.000} C_DIS
LIN {X -97.366,Y -24.270,Z -42.764,A -90.000,B 90.000,C 0.000} C_DIS
LIN {X -96.972,Y -24.234,Z -42.685,A -90.000,B 90.000,C 0.000} C_DIS
LIN {X -96.804,Y -24.221,Z -42.657,A -90.000,B 90.000,C 0.000} C_DIS
LIN {X -96.555,Y -24.186,Z -42.626,A -90.000,B 90.000,C 0.000} C_DIS
LIN {X -96.372,Y -24.165,Z -42.610,A -90.000,B 90.000,C 0.000} C_DIS
LIN {X -96.193,Y -24.147,Z -42.597,A -90.000,B 90.000,C 0.000} C_DIS
LIN {X -96.060,Y -24.136,Z -42.590,A -90.000,B 90.000,C 0.000} C_DIS
LIN {X -95.842,Y -24.122,Z -42.586,A -90.000,B 90.000,C 0.000} C_DIS
LIN {X -95.709,Y -24.111,Z -42.586,A -90.000,B 90.000,C 0.000} C_DIS
LIN {X -95.537,Y -24.100,Z -42.591,A -90.000,B 90.000,C 0.000} C_DIS
LIN {X -95.474,Y -24.097,Z -42.594,A -90.000,B 90.000,C 0.000} C_DIS
LIN {X -94.813,Y -24.050,Z -42.637,A -90.000,B 90.000,C 0.000} C_DIS
LIN {X -94.521,Y -24.023,Z -42.662,A -90.000,B 90.000,C 0.000} C_DIS
LIN {X -94.066,Y -23.987,Z -42.706,A -90.000,B 90.000,C 0.000} C_DIS
LIN {X -93.919,Y -24.020,Z -42.684,A -90.000,B 90.000,C 0.000} C_DIS
LIN {X -93.629,Y -24.089,Z -42.644,A -90.000,B 90.000,C 0.000} C_DIS
LIN {X -93.559,Y -24.102,Z -42.638,A -90.000,B 90.000,C 0.000} C_DIS
LIN {X -93.365,Y -24.138,Z -42.631,A -90.000,B 90.000,C 0.000} C_DIS
LIN {X -93.013,Y -24.216,Z -42.620,A -90.000,B 90.000,C 0.000} C_DIS
LIN {X -92.801,Y -24.264,Z -42.620,A -90.000,B 90.000,C 0.000} C_DIS
LIN {X -92.713,Y -24.284,Z -42.623,A -90.000,B 90.000,C 0.000} C_DIS
LIN {X -92.440,Y -24.347,Z -42.637,A -90.000,B 90.000,C 0.000} C_DIS
LIN {X -92.142,Y -24.415,Z -42.656,A -90.000,B 90.000,C 0.000} C_DIS
LIN {X -92.037,Y -24.440,Z -42.666,A -90.000,B 90.000,C 0.000} C_DIS
LIN {X -91.772,Y -24.502,Z -42.700,A -90.000,B 90.000,C 0.000} C_DIS
LIN {X -91.285,Y -24.616,Z -42.768,A -90.000,B 90.000,C 0.000} C_DIS
LIN {X -90.930,Y -24.700,Z -42.831,A -90.000,B 90.000,C 0.000} C_DIS
LIN {X -90.552,Y -24.790,Z -42.903,A -90.000,B 90.000,C 0.000} C_DIS
LIN {X -90.336,Y -24.841,Z -42.948,A -90.000,B 90.000,C 0.000} C_DIS
LIN {X -90.296,Y -24.824,Z -42.592,A -90.000,B 90.000,C 0.000} C_DIS
LIN {X -90.285,Y -24.824,Z -42.490,A -90.000,B 90.000,C 0.000} C_DIS
LIN {X -90.260,Y -24.820,Z -42.106,A -90.000,B 90.000,C 0.000} C_DIS
LIN {X -90.237,Y -24.807,Z -41.871,A -90.000,B 90.000,C 0.000} C_DIS
LIN {X -90.218,Y -24.797,Z -41.735,A -90.000,B 90.000,C 0.000} C_DIS
LIN {X -90.198,Y -24.791,Z -41.633,A -90.000,B 90.000,C 0.000} C_DIS
LIN {X -90.180,Y -24.787,Z -41.561,A -90.000,B 90.000,C 0.000} C_DIS
LIN {X -90.152,Y -24.784,Z -41.466,A -90.000,B 90.000,C 0.000} C_DIS
LIN {X -90.050,Y -24.782,Z -41.138,A -90.000,B 90.000,C 0.000} C_DIS
LIN {X -89.993,Y -24.783,Z -40.964,A -90.000,B 90.000,C 0.000} C_DIS
LIN {X -89.906,Y -24.771,Z -40.711,A -90.000,B 90.000,C 0.000} C_DIS
LIN {X -89.883,Y -24.768,Z -40.651,A -90.000,B 90.000,C 0.000} C_DIS
LIN {X -89.857,Y -24.765,Z -40.593,A -90.000,B 90.000,C 0.000} C_DIS
LIN {X -89.773,Y -24.759,Z -40.427,A -90.000,B 90.000,C 0.000} C_DIS
LIN {X -89.702,Y -24.756,Z -40.302,A -90.000,B 90.000,C 0.000} C_DIS
LIN {X -89.614,Y -24.744,Z -40.153,A -90.000,B 90.000,C 0.000} C_DIS
LIN {X -89.504,Y -24.744,Z -39.995,A -90.000,B 90.000,C 0.000} C_DIS
LIN {X -89.426,Y -24.747,Z -39.897,A -90.000,B 90.000,C 0.000} C_DIS
LIN {X -89.321,Y -24.730,Z -39.693,A -90.000,B 90.000,C 0.000} C_DIS
LIN {X -89.271,Y -24.726,Z -39.595,A -90.000,B 90.000,C 0.000} C_DIS
LIN {X -89.193,Y -24.715,Z -39.464,A -90.000,B 90.000,C 0.000} C_DIS
LIN {X -89.136,Y -24.709,Z -39.378,A -90.000,B 90.000,C 0.000} C_DIS
LIN {X -89.004,Y -24.684,Z -39.190,A -90.000,B 90.000,C 0.000} C_DIS
LIN {X -88.943,Y -24.673,Z -39.111,A -90.000,B 90.000,C 0.000} C_DIS
LIN {X -88.885,Y -24.665,Z -39.044,A -90.000,B 90.000,C 0.000} C_DIS
LIN {X -88.743,Y -24.649,Z -38.894,A -90.000,B 90.000,C 0.000} C_DIS
LIN {X -88.632,Y -24.648,Z -38.775,A -90.000,B 90.000,C 0.000} C_DIS
LIN {X -88.574,Y -24.644,Z -38.717,A -90.000,B 90.000,C 0.000} C_DIS
LIN {X -88.456,Y -24.639,Z -38.612,A -90.000,B 90.000,C 0.000} C_DIS
LIN {X -88.338,Y -24.633,Z -38.520,A -90.000,B 90.000,C 0.000} C_DIS
LIN {X -88.001,Y -24.618,Z -38.274,A -90.000,B 90.000,C 0.000} C_DIS
LIN {X -87.925,Y -24.612,Z -38.219,A -90.000,B 90.000,C 0.000} C_DIS
LIN {X -87.768,Y -24.598,Z -38.068,A -90.000,B 90.000,C 0.000} C_DIS
LIN {X -87.612,Y -24.590,Z -37.936,A -90.000,B 90.000,C 0.000} C_DIS
LIN {X -87.474,Y -24.585,Z -37.835,A -90.000,B 90.000,C 0.000} C_DIS
LIN {X -87.321,Y -24.578,Z -37.725,A -90.000,B 90.000,C 0.000} C_DIS
LIN {X -87.238,Y -24.574,Z -37.671,A -90.000,B 90.000,C 0.000} C_DIS
LIN {X -87.078,Y -24.565,Z -37.584,A -90.000,B 90.000,C 0.000} C_DIS
LIN {X -86.804,Y -24.556,Z -37.450,A -90.000,B 90.000,C 0.000} C_DIS
LIN {X -86.698,Y -24.548,Z -37.387,A -90.000,B 90.000,C 0.000} C_DIS
LIN {X -86.423,Y -24.535,Z -37.220,A -90.000,B 90.000,C 0.000} C_DIS
LIN {X -86.283,Y -24.525,Z -37.137,A -90.000,B 90.000,C 0.000} C_DIS
LIN {X -86.134,Y -24.518,Z -37.056,A -90.000,B 90.000,C 0.000} C_DIS
LIN {X -85.875,Y -24.512,Z -36.928,A -90.000,B 90.000,C 0.000} C_DIS
LIN {X -85.752,Y -24.511,Z -36.873,A -90.000,B 90.000,C 0.000} C_DIS
LIN {X -85.717,Y -24.511,Z -36.858,A -90.000,B 90.000,C 0.000} C_DIS
LIN {X -85.576,Y -24.515,Z -36.807,A -90.000,B 90.000,C 0.000} C_DIS
LIN {X -85.233,Y -24.529,Z -36.700,A -90.000,B 90.000,C 0.000} C_DIS
LIN {X -84.540,Y -24.533,Z -36.512,A -90.000,B 90.000,C 0.000} C_DIS
LIN {X -84.059,Y -24.530,Z -36.364,A -90.000,B 90.000,C 0.000} C_DIS
LIN {X -83.601,Y -24.529,Z -36.229,A -90.000,B 90.000,C 0.000} C_DIS
LIN {X -83.454,Y -24.532,Z -36.193,A -90.000,B 90.000,C 0.000} C_DIS
LIN {X -83.399,Y -24.534,Z -36.181,A -90.000,B 90.000,C 0.000} C_DIS
LIN {X -83.252,Y -24.532,Z -36.161,A -90.000,B 90.000,C 0.000} C_DIS
LIN {X -82.977,Y -24.532,Z -36.132,A -90.000,B 90.000,C 0.000} C_DIS
LIN {X -82.810,Y -24.534,Z -36.122,A -90.000,B 90.000,C 0.000} C_DIS
LIN {X -82.711,Y -24.536,Z -36.118,A -90.000,B 90.000,C 0.000} C_DIS
LIN {X -81.790,Y -24.574,Z -36.076,A -90.000,B 90.000,C 0.000} C_DIS
LIN {X -81.557,Y -24.580,Z -36.067,A -90.000,B 90.000,C 0.000} C_DIS
LIN {X -81.334,Y -24.572,Z -36.060,A -90.000,B 90.000,C 0.000} C_DIS
LIN {X -81.219,Y -24.567,Z -36.056,A -90.000,B 90.000,C 0.000} C_DIS
LIN {X -81.077,Y -24.566,Z -36.056,A -90.000,B 90.000,C 0.000} C_DIS
LIN {X -80.904,Y -24.566,Z -36.061,A -90.000,B 90.000,C 0.000} C_DIS
LIN {X -80.528,Y -24.573,Z -36.089,A -90.000,B 90.000,C 0.000} C_DIS
LIN {X -80.423,Y -24.579,Z -36.099,A -90.000,B 90.000,C 0.000} C_DIS
LIN {X -80.243,Y -24.589,Z -36.122,A -90.000,B 90.000,C 0.000} C_DIS
LIN {X -79.999,Y -24.598,Z -36.156,A -90.000,B 90.000,C 0.000} C_DIS
LIN {X -79.852,Y -24.596,Z -36.179,A -90.000,B 90.000,C 0.000} C_DIS
LIN {X -79.716,Y -24.600,Z -36.198,A -90.000,B 90.000,C 0.000} C_DIS
LIN {X -79.350,Y -24.590,Z -36.257,A -90.000,B 90.000,C 0.000} C_DIS
LIN {X -79.109,Y -24.588,Z -36.293,A -90.000,B 90.000,C 0.000} C_DIS
LIN {X -78.984,Y -24.586,Z -36.310,A -90.000,B 90.000,C 0.000} C_DIS
LIN {X -78.777,Y -24.584,Z -36.343,A -90.000,B 90.000,C 0.000} C_DIS
LIN {X -78.588,Y -24.584,Z -36.379,A -90.000,B 90.000,C 0.000} C_DIS
LIN {X -78.200,Y -24.591,Z -36.473,A -90.000,B 90.000,C 0.000} C_DIS
LIN {X -77.864,Y -24.593,Z -36.561,A -90.000,B 90.000,C 0.000} C_DIS
LIN {X -76.609,Y -24.569,Z -36.903,A -90.000,B 90.000,C 0.000} C_DIS
LIN {X -76.166,Y -24.567,Z -37.038,A -90.000,B 90.000,C 0.000} C_DIS
LIN {X -75.928,Y -24.563,Z -37.113,A -90.000,B 90.000,C 0.000} C_DIS
LIN {X -75.009,Y -24.566,Z -37.395,A -90.000,B 90.000,C 0.000} C_DIS
LIN {X -74.739,Y -24.564,Z -37.469,A -90.000,B 90.000,C 0.000} C_DIS
LIN {X -73.937,Y -24.550,Z -37.690,A -90.000,B 90.000,C 0.000} C_DIS
LIN {X -73.235,Y -24.545,Z -37.882,A -90.000,B 90.000,C 0.000} C_DIS
LIN {X -72.772,Y -24.531,Z -38.015,A -90.000,B 90.000,C 0.000} C_DIS
LIN {X -72.131,Y -24.520,Z -38.191,A -90.000,B 90.000,C 0.000} C_DIS
LIN {X -71.687,Y -24.519,Z -38.328,A -90.000,B 90.000,C 0.000} C_DIS
LIN {X -71.400,Y -24.519,Z -38.417,A -90.000,B 90.000,C 0.000} C_DIS
LIN {X -70.498,Y -24.497,Z -38.706,A -90.000,B 90.000,C 0.000} C_DIS
LIN {X -70.393,Y -24.496,Z -38.742,A -90.000,B 90.000,C 0.000} C_DIS
LIN {X -69.606,Y -24.497,Z -39.035,A -90.000,B 90.000,C 0.000} C_DIS
LIN {X -68.939,Y -24.484,Z -39.291,A -90.000,B 90.000,C 0.000} C_DIS
LIN {X -68.609,Y -24.476,Z -39.418,A -90.000,B 90.000,C 0.000} C_DIS
LIN {X -68.261,Y -24.473,Z -39.565,A -90.000,B 90.000,C 0.000} C_DIS
LIN {X -66.823,Y -24.471,Z -40.205,A -90.000,B 90.000,C 0.000} C_DIS
LIN {X -66.118,Y -24.469,Z -40.520,A -90.000,B 90.000,C 0.000} C_DIS
LIN {X -65.576,Y -24.468,Z -40.769,A -90.000,B 90.000,C 0.000} C_DIS
LIN {X -64.838,Y -24.468,Z -41.113,A -90.000,B 90.000,C 0.000} C_DIS
LIN {X -63.804,Y -24.479,Z -41.589,A -90.000,B 90.000,C 0.000} C_DIS
LIN {X -63.451,Y -24.479,Z -41.744,A -90.000,B 90.000,C 0.000} C_DIS
LIN {X -62.423,Y -24.475,Z -42.197,A -90.000,B 90.000,C 0.000} C_DIS
LIN {X -61.558,Y -24.490,Z -42.570,A -90.000,B 90.000,C 0.000} C_DIS
LIN {X -61.145,Y -24.488,Z -42.728,A -90.000,B 90.000,C 0.000} C_DIS
LIN {X -59.902,Y -24.473,Z -43.208,A -90.000,B 90.000,C 0.000} C_DIS
LIN {X -59.009,Y -24.485,Z -43.543,A -90.000,B 90.000,C 0.000} C_DIS
LIN {X -58.174,Y -24.469,Z -43.798,A -90.000,B 90.000,C 0.000} C_DIS
LIN {X -57.174,Y -24.458,Z -44.101,A -90.000,B 90.000,C 0.000} C_DIS
LIN {X -56.801,Y -24.458,Z -44.212,A -90.000,B 90.000,C 0.000} C_DIS
LIN {X -56.433,Y -24.461,Z -44.324,A -90.000,B 90.000,C 0.000} C_DIS
LIN {X -55.232,Y -24.431,Z -44.613,A -90.000,B 90.000,C 0.000} C_DIS
LIN {X -54.367,Y -24.412,Z -44.834,A -90.000,B 90.000,C 0.000} C_DIS
LIN {X -53.985,Y -24.411,Z -44.929,A -90.000,B 90.000,C 0.000} C_DIS
LIN {X -53.478,Y -24.393,Z -45.024,A -90.000,B 90.000,C 0.000} C_DIS
LIN {X -52.810,Y -24.377,Z -45.162,A -90.000,B 90.000,C 0.000} C_DIS
LIN {X -52.524,Y -24.368,Z -45.224,A -90.000,B 90.000,C 0.000} C_DIS
LIN {X -51.417,Y -24.353,Z -45.493,A -90.000,B 90.000,C 0.000} C_DIS
LIN {X -51.088,Y -24.352,Z -45.572,A -90.000,B 90.000,C 0.000} C_DIS
LIN {X -50.360,Y -24.340,Z -45.731,A -90.000,B 90.000,C 0.000} C_DIS
LIN {X -48.719,Y -24.319,Z -46.080,A -90.000,B 90.000,C 0.000} C_DIS
LIN {X -48.142,Y -24.319,Z -46.199,A -90.000,B 90.000,C 0.000} C_DIS
LIN {X -47.085,Y -24.299,Z -46.398,A -90.000,B 90.000,C 0.000} C_DIS
LIN {X -45.912,Y -24.285,Z -46.629,A -90.000,B 90.000,C 0.000} C_DIS
LIN {X -45.705,Y -24.281,Z -46.672,A -90.000,B 90.000,C 0.000} C_DIS
LIN {X -45.238,Y -24.280,Z -46.765,A -90.000,B 90.000,C 0.000} C_DIS
LIN {X -45.085,Y -24.281,Z -46.797,A -90.000,B 90.000,C 0.000} C_DIS
LIN {X -44.264,Y -24.277,Z -46.956,A -90.000,B 90.000,C 0.000} C_DIS
LIN {X -44.017,Y -24.274,Z -47.005,A -90.000,B 90.000,C 0.000} C_DIS
LIN {X -43.344,Y -24.264,Z -47.140,A -90.000,B 90.000,C 0.000} C_DIS
LIN {X -42.655,Y -24.258,Z -47.283,A -90.000,B 90.000,C 0.000} C_DIS
LIN {X -42.285,Y -24.258,Z -47.357,A -90.000,B 90.000,C 0.000} C_DIS
LIN {X -42.083,Y -24.256,Z -47.399,A -90.000,B 90.000,C 0.000} C_DIS
LIN {X -41.372,Y -24.246,Z -47.540,A -90.000,B 90.000,C 0.000} C_DIS
LIN {X -40.063,Y -24.235,Z -47.806,A -90.000,B 90.000,C 0.000} C_DIS
LIN {X -39.354,Y -24.218,Z -47.960,A -90.000,B 90.000,C 0.000} C_DIS
LIN {X -38.772,Y -24.214,Z -48.091,A -90.000,B 90.000,C 0.000} C_DIS
LIN {X -37.473,Y -24.200,Z -48.377,A -90.000,B 90.000,C 0.000} C_DIS
LIN {X -37.260,Y -24.197,Z -48.426,A -90.000,B 90.000,C 0.000} C_DIS
LIN {X -36.927,Y -24.189,Z -48.505,A -90.000,B 90.000,C 0.000} C_DIS
LIN {X -36.156,Y -24.175,Z -48.697,A -90.000,B 90.000,C 0.000} C_DIS
LIN {X -35.519,Y -24.159,Z -48.859,A -90.000,B 90.000,C 0.000} C_DIS
LIN {X -33.601,Y -24.129,Z -49.369,A -90.000,B 90.000,C 0.000} C_DIS
LIN {X -33.040,Y -24.116,Z -49.514,A -90.000,B 90.000,C 0.000} C_DIS
LIN {X -32.436,Y -24.097,Z -49.677,A -90.000,B 90.000,C 0.000} C_DIS
LIN {X -29.709,Y -24.041,Z -50.451,A -90.000,B 90.000,C 0.000} C_DIS
LIN {X -29.177,Y -24.025,Z -50.606,A -90.000,B 90.000,C 0.000} C_DIS
LIN {X -27.333,Y -23.988,Z -51.160,A -90.000,B 90.000,C 0.000} C_DIS
LIN {X -26.962,Y -23.983,Z -51.269,A -90.000,B 90.000,C 0.000} C_DIS
LIN {X -25.902,Y -23.960,Z -51.570,A -90.000,B 90.000,C 0.000} C_DIS
LIN {X -25.036,Y -23.940,Z -51.818,A -90.000,B 90.000,C 0.000} C_DIS
LIN {X -24.769,Y -23.937,Z -51.892,A -90.000,B 90.000,C 0.000} C_DIS
LIN {X -23.716,Y -23.912,Z -52.166,A -90.000,B 90.000,C 0.000} C_DIS
LIN {X -23.199,Y -23.891,Z -52.310,A -90.000,B 90.000,C 0.000} C_DIS
LIN {X -23.051,Y -23.891,Z -52.344,A -90.000,B 90.000,C 0.000} C_DIS
LIN {X -22.677,Y -23.888,Z -52.424,A -90.000,B 90.000,C 0.000} C_DIS
LIN {X -22.357,Y -23.878,Z -52.488,A -90.000,B 90.000,C 0.000} C_DIS
LIN {X -21.908,Y -23.858,Z -52.585,A -90.000,B 90.000,C 0.000} C_DIS
LIN {X -21.788,Y -23.857,Z -52.598,A -90.000,B 90.000,C 0.000} C_DIS
LIN {X -21.483,Y -23.853,Z -52.632,A -90.000,B 90.000,C 0.000} C_DIS
LIN {X -21.080,Y -23.835,Z -52.675,A -90.000,B 90.000,C 0.000} C_DIS
LIN {X -20.935,Y -23.818,Z -52.682,A -90.000,B 90.000,C 0.000} C_DIS
LIN {X -20.594,Y -23.805,Z -52.665,A -90.000,B 90.000,C 0.000} C_DIS
LIN {X -20.567,Y -23.802,Z -52.662,A -90.000,B 90.000,C 0.000} C_DIS
LIN {X -20.229,Y -23.851,Z -52.521,A -90.000,B 90.000,C 0.000} C_DIS
LIN {X -20.042,Y -23.877,Z -52.449,A -90.000,B 90.000,C 0.000} C_DIS
LIN {X -19.766,Y -23.913,Z -52.357,A -90.000,B 90.000,C 0.000} C_DIS
LIN {X -19.397,Y -23.970,Z -52.178,A -90.000,B 90.000,C 0.000} C_DIS
LIN {X -18.936,Y -24.040,Z -51.974,A -90.000,B 90.000,C 0.000} C_DIS
LIN {X -18.648,Y -24.085,Z -51.830,A -90.000,B 90.000,C 0.000} C_DIS
LIN {X -18.252,Y -24.129,Z -51.649,A -90.000,B 90.000,C 0.000} C_DIS
LIN {X -17.685,Y -24.192,Z -51.396,A -90.000,B 90.000,C 0.000} C_DIS
LIN {X -17.396,Y -24.225,Z -51.276,A -90.000,B 90.000,C 0.000} C_DIS
LIN {X -17.240,Y -24.245,Z -51.210,A -90.000,B 90.000,C 0.000} C_DIS
LIN {X -17.095,Y -24.260,Z -51.152,A -90.000,B 90.000,C 0.000} C_DIS
LIN {X -16.318,Y -24.323,Z -50.854,A -90.000,B 90.000,C 0.000} C_DIS
LIN {X -15.956,Y -24.354,Z -50.725,A -90.000,B 90.000,C 0.000} C_DIS
LIN {X -15.805,Y -24.366,Z -50.676,A -90.000,B 90.000,C 0.000} C_DIS
LIN {X -15.691,Y -24.376,Z -50.644,A -90.000,B 90.000,C 0.000} C_DIS
LIN {X -15.575,Y -24.385,Z -50.617,A -90.000,B 90.000,C 0.000} C_DIS
LIN {X -15.223,Y -24.414,Z -50.523,A -90.000,B 90.000,C 0.000} C_DIS
LIN {X -14.601,Y -24.444,Z -50.371,A -90.000,B 90.000,C 0.000} C_DIS
LIN {X -14.108,Y -24.477,Z -50.260,A -90.000,B 90.000,C 0.000} C_DIS
LIN {X -13.393,Y -24.525,Z -50.122,A -90.000,B 90.000,C 0.000} C_DIS
LIN {X -13.115,Y -24.540,Z -50.071,A -90.000,B 90.000,C 0.000} C_DIS
LIN {X -12.915,Y -24.548,Z -50.039,A -90.000,B 90.000,C 0.000} C_DIS
LIN {X -12.783,Y -24.553,Z -50.025,A -90.000,B 90.000,C 0.000} C_DIS
LIN {X -11.857,Y -24.585,Z -49.912,A -90.000,B 90.000,C 0.000} C_DIS
LIN {X -10.975,Y -24.629,Z -49.843,A -90.000,B 90.000,C 0.000} C_DIS
LIN {X -10.641,Y -24.637,Z -49.821,A -90.000,B 90.000,C 0.000} C_DIS
LIN {X -10.334,Y -24.641,Z -49.798,A -90.000,B 90.000,C 0.000} C_DIS
LIN {X -9.960,Y -24.648,Z -49.779,A -90.000,B 90.000,C 0.000} C_DIS
LIN {X -9.027,Y -24.669,Z -49.752,A -90.000,B 90.000,C 0.000} C_DIS
LIN {X -8.978,Y -24.671,Z -49.753,A -90.000,B 90.000,C 0.000} C_DIS
LIN {X -8.746,Y -24.675,Z -49.751,A -90.000,B 90.000,C 0.000} C_DIS
LIN {X -8.229,Y -24.674,Z -49.751,A -90.000,B 90.000,C 0.000} C_DIS
LIN {X -6.030,Y -24.678,Z -49.802,A -90.000,B 90.000,C 0.000} C_DIS
LIN {X -5.526,Y -24.672,Z -49.824,A -90.000,B 90.000,C 0.000} C_DIS
LIN {X -5.211,Y -24.669,Z -49.843,A -90.000,B 90.000,C 0.000} C_DIS
LIN {X -3.937,Y -24.643,Z -49.923,A -90.000,B 90.000,C 0.000} C_DIS
LIN {X -3.443,Y -24.629,Z -49.953,A -90.000,B 90.000,C 0.000} C_DIS
LIN {X -3.164,Y -24.624,Z -49.979,A -90.000,B 90.000,C 0.000} C_DIS
LIN {X -2.691,Y -24.611,Z -50.006,A -90.000,B 90.000,C 0.000} C_DIS
LIN {X -2.081,Y -24.596,Z -50.054,A -90.000,B 90.000,C 0.000} C_DIS
LIN {X -1.683,Y -24.583,Z -50.086,A -90.000,B 90.000,C 0.000} C_DIS
LIN {X -1.459,Y -24.573,Z -50.106,A -90.000,B 90.000,C 0.000} C_DIS
LIN {X -0.541,Y -24.543,Z -50.182,A -90.000,B 90.000,C 0.000} C_DIS
LIN {X -0.176,Y -24.534,Z -50.219,A -90.000,B 90.000,C 0.000} C_DIS
LIN {X 0.196,Y -24.515,Z -50.234,A -90.000,B 90.000,C 0.000} C_DIS
LIN {X 0.376,Y -24.510,Z -50.240,A -90.000,B 90.000,C 0.000} C_DIS
LIN {X 0.689,Y -24.500,Z -50.253,A -90.000,B 90.000,C 0.000} C_DIS
LIN {X 1.117,Y -24.488,Z -50.273,A -90.000,B 90.000,C 0.000} C_DIS
LIN {X 1.537,Y -24.464,Z -50.268,A -90.000,B 90.000,C 0.000} C_DIS
LIN {X 2.215,Y -24.402,Z -50.274,A -90.000,B 90.000,C 0.000} C_DIS
LIN {X 2.311,Y -24.396,Z -50.272,A -90.000,B 90.000,C 0.000} C_DIS
LIN {X 3.078,Y -24.338,Z -50.241,A -90.000,B 90.000,C 0.000} C_DIS
LIN {X 3.221,Y -24.322,Z -50.239,A -90.000,B 90.000,C 0.000} C_DIS
LIN {X 3.620,Y -24.278,Z -50.239,A -90.000,B 90.000,C 0.000} C_DIS
LIN {X 4.109,Y -24.231,Z -50.249,A -90.000,B 90.000,C 0.000} C_DIS
LIN {X 4.488,Y -24.207,Z -50.249,A -90.000,B 90.000,C 0.000} C_DIS
LIN {X 4.824,Y -24.174,Z -50.264,A -90.000,B 90.000,C 0.000} C_DIS
LIN {X 4.992,Y -24.162,Z -50.277,A -90.000,B 90.000,C 0.000} C_DIS
LIN {X 5.811,Y -24.095,Z -50.335,A -90.000,B 90.000,C 0.000} C_DIS
LIN {X 6.052,Y -24.079,Z -50.352,A -90.000,B 90.000,C 0.000} C_DIS
LIN {X 6.206,Y -24.071,Z -50.364,A -90.000,B 90.000,C 0.000} C_DIS
LIN {X 6.589,Y -24.042,Z -50.403,A -90.000,B 90.000,C 0.000} C_DIS
LIN {X 7.422,Y -23.987,Z -50.498,A -90.000,B 90.000,C 0.000} C_DIS
LIN {X 7.540,Y -23.975,Z -50.516,A -90.000,B 90.000,C 0.000} C_DIS
LIN {X 8.683,Y -23.888,Z -50.664,A -90.000,B 90.000,C 0.000} C_DIS
LIN {X 8.935,Y -23.872,Z -50.704,A -90.000,B 90.000,C 0.000} C_DIS
LIN {X 9.772,Y -23.816,Z -50.849,A -90.000,B 90.000,C 0.000} C_DIS
LIN {X 10.200,Y -23.798,Z -50.931,A -90.000,B 90.000,C 0.000} C_DIS
LIN {X 10.516,Y -23.788,Z -50.998,A -90.000,B 90.000,C 0.000} C_DIS
LIN {X 10.904,Y -23.770,Z -51.087,A -90.000,B 90.000,C 0.000} C_DIS
LIN {X 11.201,Y -23.764,Z -51.159,A -90.000,B 90.000,C 0.000} C_DIS
LIN {X 12.397,Y -23.749,Z -51.457,A -90.000,B 90.000,C 0.000} C_DIS
LIN {X 12.778,Y -23.746,Z -51.549,A -90.000,B 90.000,C 0.000} C_DIS
LIN {X 12.984,Y -23.812,Z -51.516,A -90.000,B 90.000,C 0.000} C_DIS
LIN {X 13.179,Y -23.875,Z -51.485,A -90.000,B 90.000,C 0.000} C_DIS
LIN {X 13.396,Y -23.962,Z -51.441,A -90.000,B 90.000,C 0.000} C_DIS
LIN {X 13.544,Y -24.022,Z -51.416,A -90.000,B 90.000,C 0.000} C_DIS
LIN {X 13.849,Y -24.136,Z -51.383,A -90.000,B 90.000,C 0.000} C_DIS
LIN {X 14.060,Y -24.223,Z -51.365,A -90.000,B 90.000,C 0.000} C_DIS
LIN {X 14.355,Y -24.335,Z -51.354,A -90.000,B 90.000,C 0.000} C_DIS
LIN {X 14.477,Y -24.382,Z -51.351,A -90.000,B 90.000,C 0.000} C_DIS
LIN {X 14.562,Y -24.385,Z -51.227,A -90.000,B 90.000,C 0.000} C_DIS
LIN {X 14.756,Y -24.395,Z -50.956,A -90.000,B 90.000,C 0.000} C_DIS
LIN {X 15.100,Y -24.399,Z -50.487,A -90.000,B 90.000,C 0.000} C_DIS
LIN {X 15.295,Y -24.392,Z -50.237,A -90.000,B 90.000,C 0.000} C_DIS
LIN {X 15.396,Y -24.383,Z -50.111,A -90.000,B 90.000,C 0.000} C_DIS
LIN {X 15.509,Y -24.377,Z -49.981,A -90.000,B 90.000,C 0.000} C_DIS
LIN {X 15.717,Y -24.377,Z -49.773,A -90.000,B 90.000,C 0.000} C_DIS
LIN {X 16.100,Y -24.361,Z -49.409,A -90.000,B 90.000,C 0.000} C_DIS
LIN {X 16.256,Y -24.348,Z -49.265,A -90.000,B 90.000,C 0.000} C_DIS
LIN {X 16.636,Y -24.337,Z -48.933,A -90.000,B 90.000,C 0.000} C_DIS
LIN {X 16.811,Y -24.325,Z -48.785,A -90.000,B 90.000,C 0.000} C_DIS
LIN {X 16.914,Y -24.320,Z -48.702,A -90.000,B 90.000,C 0.000} C_DIS
LIN {X 17.113,Y -24.316,Z -48.556,A -90.000,B 90.000,C 0.000} C_DIS
LIN {X 17.628,Y -24.283,Z -48.187,A -90.000,B 90.000,C 0.000} C_DIS
LIN {X 17.998,Y -24.269,Z -47.926,A -90.000,B 90.000,C 0.000} C_DIS
LIN {X 18.063,Y -24.268,Z -47.882,A -90.000,B 90.000,C 0.000} C_DIS
LIN {X 18.339,Y -24.251,Z -47.703,A -90.000,B 90.000,C 0.000} C_DIS
LIN {X 18.763,Y -24.203,Z -47.446,A -90.000,B 90.000,C 0.000} C_DIS
LIN {X 18.807,Y -24.199,Z -47.420,A -90.000,B 90.000,C 0.000} C_DIS
LIN {X 18.993,Y -24.188,Z -47.309,A -90.000,B 90.000,C 0.000} C_DIS
LIN {X 19.442,Y -24.160,Z -47.039,A -90.000,B 90.000,C 0.000} C_DIS
LIN {X 19.886,Y -24.119,Z -46.822,A -90.000,B 90.000,C 0.000} C_DIS
LIN {X 19.998,Y -24.110,Z -46.767,A -90.000,B 90.000,C 0.000} C_DIS
LIN {X 20.355,Y -24.067,Z -46.573,A -90.000,B 90.000,C 0.000} C_DIS
LIN {X 20.469,Y -24.055,Z -46.516,A -90.000,B 90.000,C 0.000} C_DIS
LIN {X 20.643,Y -24.041,Z -46.435,A -90.000,B 90.000,C 0.000} C_DIS
LIN {X 21.013,Y -23.997,Z -46.277,A -90.000,B 90.000,C 0.000} C_DIS
LIN {X 21.406,Y -23.948,Z -46.125,A -90.000,B 90.000,C 0.000} C_DIS
LIN {X 21.436,Y -23.944,Z -46.115,A -90.000,B 90.000,C 0.000} C_DIS
LIN {X 21.982,Y -23.918,Z -45.886,A -90.000,B 90.000,C 0.000} C_DIS
LIN {X 22.230,Y -23.897,Z -45.791,A -90.000,B 90.000,C 0.000} C_DIS
LIN {X 22.353,Y -23.884,Z -45.743,A -90.000,B 90.000,C 0.000} C_DIS
LIN {X 22.654,Y -23.849,Z -45.629,A -90.000,B 90.000,C 0.000} C_DIS
LIN {X 23.179,Y -23.790,Z -45.447,A -90.000,B 90.000,C 0.000} C_DIS
LIN {X 23.476,Y -23.763,Z -45.345,A -90.000,B 90.000,C 0.000} C_DIS
LIN {X 23.627,Y -23.750,Z -45.295,A -90.000,B 90.000,C 0.000} C_DIS
LIN {X 23.715,Y -23.741,Z -45.272,A -90.000,B 90.000,C 0.000} C_DIS
LIN {X 23.925,Y -23.732,Z -45.200,A -90.000,B 90.000,C 0.000} C_DIS
LIN {X 24.112,Y -23.717,Z -45.144,A -90.000,B 90.000,C 0.000} C_DIS
LIN {X 24.219,Y -23.708,Z -45.111,A -90.000,B 90.000,C 0.000} C_DIS
LIN {X 24.855,Y -23.663,Z -44.898,A -90.000,B 90.000,C 0.000} C_DIS
LIN {X 25.079,Y -23.638,Z -44.839,A -90.000,B 90.000,C 0.000} C_DIS
LIN {X 25.235,Y -23.624,Z -44.800,A -90.000,B 90.000,C 0.000} C_DIS
LIN {X 25.654,Y -23.594,Z -44.702,A -90.000,B 90.000,C 0.000} C_DIS
LIN {X 25.863,Y -23.587,Z -44.640,A -90.000,B 90.000,C 0.000} C_DIS
LIN {X 26.031,Y -23.577,Z -44.588,A -90.000,B 90.000,C 0.000} C_DIS
LIN {X 26.287,Y -23.562,Z -44.516,A -90.000,B 90.000,C 0.000} C_DIS
LIN {X 26.428,Y -23.555,Z -44.477,A -90.000,B 90.000,C 0.000} C_DIS
LIN {X 26.809,Y -23.528,Z -44.392,A -90.000,B 90.000,C 0.000} C_DIS
LIN {X 27.395,Y -23.508,Z -44.252,A -90.000,B 90.000,C 0.000} C_DIS
LIN {X 27.880,Y -23.485,Z -44.153,A -90.000,B 90.000,C 0.000} C_DIS
LIN {X 28.152,Y -23.478,Z -44.084,A -90.000,B 90.000,C 0.000} C_DIS
LIN {X 28.382,Y -23.475,Z -44.028,A -90.000,B 90.000,C 0.000} C_DIS
LIN {X 28.471,Y -23.472,Z -44.010,A -90.000,B 90.000,C 0.000} C_DIS
LIN {X 28.800,Y -23.471,Z -43.925,A -90.000,B 90.000,C 0.000} C_DIS
LIN {X 29.453,Y -23.466,Z -43.763,A -90.000,B 90.000,C 0.000} C_DIS
LIN {X 29.515,Y -23.467,Z -43.749,A -90.000,B 90.000,C 0.000} C_DIS
LIN {X 30.242,Y -23.496,Z -43.560,A -90.000,B 90.000,C 0.000} C_DIS
LIN {X 30.786,Y -23.521,Z -43.405,A -90.000,B 90.000,C 0.000} C_DIS
LIN {X 30.878,Y -23.527,Z -43.380,A -90.000,B 90.000,C 0.000} C_DIS
LIN {X 31.316,Y -23.562,Z -43.256,A -90.000,B 90.000,C 0.000} C_DIS
LIN {X 31.791,Y -23.596,Z -43.118,A -90.000,B 90.000,C 0.000} C_DIS
LIN {X 32.306,Y -23.649,Z -42.982,A -90.000,B 90.000,C 0.000} C_DIS
LIN {X 32.397,Y -23.658,Z -42.958,A -90.000,B 90.000,C 0.000} C_DIS
LIN {X 32.448,Y -23.662,Z -42.944,A -90.000,B 90.000,C 0.000} C_DIS
LIN {X 32.919,Y -23.707,Z -42.817,A -90.000,B 90.000,C 0.000} C_DIS
LIN {X 33.130,Y -23.716,Z -42.750,A -90.000,B 90.000,C 0.000} C_DIS
LIN {X 33.451,Y -23.721,Z -42.635,A -90.000,B 90.000,C 0.000} C_DIS
LIN {X 34.395,Y -23.728,Z -42.306,A -90.000,B 90.000,C 0.000} C_DIS
LIN {X 35.461,Y -23.719,Z -41.917,A -90.000,B 90.000,C 0.000} C_DIS
LIN {X 35.761,Y -23.711,Z -41.815,A -90.000,B 90.000,C 0.000} C_DIS
LIN {X 36.166,Y -23.699,Z -41.681,A -90.000,B 90.000,C 0.000} C_DIS
LIN {X 36.791,Y -23.683,Z -41.493,A -90.000,B 90.000,C 0.000} C_DIS
LIN {X 37.460,Y -23.668,Z -41.288,A -90.000,B 90.000,C 0.000} C_DIS
LIN {X 38.135,Y -23.634,Z -41.109,A -90.000,B 90.000,C 0.000} C_DIS
LIN {X 38.675,Y -23.617,Z -40.974,A -90.000,B 90.000,C 0.000} C_DIS
LIN {X 38.875,Y -23.617,Z -40.928,A -90.000,B 90.000,C 0.000} C_DIS
LIN {X 39.338,Y -23.610,Z -40.829,A -90.000,B 90.000,C 0.000} C_DIS
LIN {X 39.995,Y -23.580,Z -40.727,A -90.000,B 90.000,C 0.000} C_DIS
LIN {X 40.539,Y -23.557,Z -40.646,A -90.000,B 90.000,C 0.000} C_DIS
LIN {X 41.139,Y -23.548,Z -40.568,A -90.000,B 90.000,C 0.000} C_DIS
LIN {X 41.667,Y -23.529,Z -40.522,A -90.000,B 90.000,C 0.000} C_DIS
LIN {X 42.461,Y -23.499,Z -40.483,A -90.000,B 90.000,C 0.000} C_DIS
LIN {X 42.583,Y -23.497,Z -40.478,A -90.000,B 90.000,C 0.000} C_DIS
LIN {X 42.919,Y -23.488,Z -40.474,A -90.000,B 90.000,C 0.000} C_DIS
LIN {X 43.108,Y -23.487,Z -40.473,A -90.000,B 90.000,C 0.000} C_DIS
LIN {X 43.591,Y -23.483,Z -40.481,A -90.000,B 90.000,C 0.000} C_DIS
LIN {X 44.059,Y -23.475,Z -40.501,A -90.000,B 90.000,C 0.000} C_DIS
LIN {X 44.149,Y -23.472,Z -40.508,A -90.000,B 90.000,C 0.000} C_DIS
LIN {X 44.368,Y -23.461,Z -40.534,A -90.000,B 90.000,C 0.000} C_DIS
LIN {X 44.897,Y -23.440,Z -40.600,A -90.000,B 90.000,C 0.000} C_DIS
LIN {X 45.452,Y -23.433,Z -40.674,A -90.000,B 90.000,C 0.000} C_DIS
LIN {X 45.917,Y -23.425,Z -40.743,A -90.000,B 90.000,C 0.000} C_DIS
LIN {X 46.685,Y -23.400,Z -40.906,A -90.000,B 90.000,C 0.000} C_DIS
LIN {X 47.192,Y -23.390,Z -41.014,A -90.000,B 90.000,C 0.000} C_DIS
LIN {X 47.679,Y -23.392,Z -41.127,A -90.000,B 90.000,C 0.000} C_DIS
LIN {X 48.032,Y -23.392,Z -41.222,A -90.000,B 90.000,C 0.000} C_DIS
LIN {X 48.141,Y -23.392,Z -41.253,A -90.000,B 90.000,C 0.000} C_DIS
LIN {X 48.727,Y -23.383,Z -41.458,A -90.000,B 90.000,C 0.000} C_DIS
LIN {X 49.310,Y -23.369,Z -41.687,A -90.000,B 90.000,C 0.000} C_DIS
LIN {X 50.387,Y -23.358,Z -42.113,A -90.000,B 90.000,C 0.000} C_DIS
LIN {X 51.087,Y -23.350,Z -42.416,A -90.000,B 90.000,C 0.000} C_DIS
LIN {X 51.451,Y -23.351,Z -42.575,A -90.000,B 90.000,C 0.000} C_DIS
LIN {X 51.925,Y -23.348,Z -42.824,A -90.000,B 90.000,C 0.000} C_DIS
LIN {X 52.483,Y -23.343,Z -43.121,A -90.000,B 90.000,C 0.000} C_DIS
LIN {X 53.144,Y -23.338,Z -43.486,A -90.000,B 90.000,C 0.000} C_DIS
LIN {X 53.851,Y -23.335,Z -43.880,A -90.000,B 90.000,C 0.000} C_DIS
LIN {X 54.260,Y -23.335,Z -44.109,A -90.000,B 90.000,C 0.000} C_DIS
LIN {X 54.547,Y -23.339,Z -44.271,A -90.000,B 90.000,C 0.000} C_DIS
LIN {X 55.018,Y -23.339,Z -44.590,A -90.000,B 90.000,C 0.000} C_DIS
LIN {X 56.603,Y -23.329,Z -45.734,A -90.000,B 90.000,C 0.000} C_DIS
LIN {X 57.160,Y -23.328,Z -46.129,A -90.000,B 90.000,C 0.000} C_DIS
LIN {X 57.351,Y -23.330,Z -46.265,A -90.000,B 90.000,C 0.000} C_DIS
LIN {X 57.765,Y -23.330,Z -46.612,A -90.000,B 90.000,C 0.000} C_DIS
LIN {X 59.334,Y -23.327,Z -47.953,A -90.000,B 90.000,C 0.000} C_DIS
LIN {X 59.861,Y -23.327,Z -48.410,A -90.000,B 90.000,C 0.000} C_DIS
LIN {X 61.118,Y -23.329,Z -49.591,A -90.000,B 90.000,C 0.000} C_DIS
LIN {X 61.772,Y -23.329,Z -50.213,A -90.000,B 90.000,C 0.000} C_DIS
LIN {X 62.063,Y -23.330,Z -50.480,A -90.000,B 90.000,C 0.000} C_DIS
LIN {X 63.581,Y -23.333,Z -51.914,A -90.000,B 90.000,C 0.000} C_DIS
LIN {X 64.245,Y -23.336,Z -52.461,A -90.000,B 90.000,C 0.000} C_DIS
LIN {X 65.154,Y -23.340,Z -53.219,A -90.000,B 90.000,C 0.000} C_DIS
LIN {X 65.205,Y -23.340,Z -53.263,A -90.000,B 90.000,C 0.000} C_DIS
LIN {X 65.402,Y -23.345,Z -53.403,A -90.000,B 90.000,C 0.000} C_DIS
LIN {X 65.567,Y -23.346,Z -53.516,A -90.000,B 90.000,C 0.000} C_DIS
LIN {X 66.067,Y -23.351,Z -53.852,A -90.000,B 90.000,C 0.000} C_DIS
LIN {X 66.886,Y -23.355,Z -54.402,A -90.000,B 90.000,C 0.000} C_DIS
LIN {X 67.582,Y -23.364,Z -54.830,A -90.000,B 90.000,C 0.000} C_DIS
LIN {X 69.343,Y -23.372,Z -55.911,A -90.000,B 90.000,C 0.000} C_DIS
LIN {X 71.094,Y -23.381,Z -56.990,A -90.000,B 90.000,C 0.000} C_DIS
LIN {X 71.541,Y -23.379,Z -57.289,A -90.000,B 90.000,C 0.000} C_DIS
LIN {X 72.671,Y -23.387,Z -58.067,A -90.000,B 90.000,C 0.000} C_DIS
LIN {X 73.205,Y -23.391,Z -58.434,A -90.000,B 90.000,C 0.000} C_DIS
LIN {X 73.343,Y -23.393,Z -58.527,A -90.000,B 90.000,C 0.000} C_DIS
LIN {X 73.454,Y -23.391,Z -58.614,A -90.000,B 90.000,C 0.000} C_DIS
LIN {X 73.847,Y -23.389,Z -58.936,A -90.000,B 90.000,C 0.000} C_DIS
LIN {X 74.168,Y -23.394,Z -59.206,A -90.000,B 90.000,C 0.000} C_DIS
LIN {X 74.784,Y -23.400,Z -59.743,A -90.000,B 90.000,C 0.000} C_DIS
LIN {X 75.324,Y -23.410,Z -60.216,A -90.000,B 90.000,C 0.000} C_DIS
LIN {X 75.803,Y -23.408,Z -60.696,A -90.000,B 90.000,C 0.000} C_DIS
LIN {X 75.989,Y -23.411,Z -60.894,A -90.000,B 90.000,C 0.000} C_DIS
LIN {X 76.367,Y -23.416,Z -61.301,A -90.000,B 90.000,C 0.000} C_DIS
LIN {X 76.908,Y -23.431,Z -61.886,A -90.000,B 90.000,C 0.000} C_DIS
LIN {X 77.015,Y -23.432,Z -62.010,A -90.000,B 90.000,C 0.000} C_DIS
LIN {X 77.354,Y -23.429,Z -62.427,A -90.000,B 90.000,C 0.000} C_DIS
LIN {X 77.897,Y -23.438,Z -63.122,A -90.000,B 90.000,C 0.000} C_DIS
LIN {X 78.161,Y -23.447,Z -63.463,A -90.000,B 90.000,C 0.000} C_DIS
LIN {X 78.283,Y -23.450,Z -63.625,A -90.000,B 90.000,C 0.000} C_DIS
LIN {X 78.335,Y -23.424,Z -63.677,A -90.000,B 90.000,C 0.000} C_DIS
LIN {X 78.412,Y -23.392,Z -63.761,A -90.000,B 90.000,C 0.000} C_DIS
LIN {X 78.480,Y -23.368,Z -63.837,A -90.000,B 90.000,C 0.000} C_DIS
LIN {X 78.547,Y -23.349,Z -63.915,A -90.000,B 90.000,C 0.000} C_DIS
LIN {X 78.627,Y -23.330,Z -64.016,A -90.000,B 90.000,C 0.000} C_DIS
LIN {X 78.846,Y -23.308,Z -64.316,A -90.000,B 90.000,C 0.000} C_DIS
LIN {X 78.850,Y -25.979,Z -64.321,A -90.000,B 90.000,C 0.000} C_DIS
LIN {X 78.861,Y -26.194,Z -64.337,A -90.000,B 90.000,C 0.000} C_DIS
LIN {X 78.906,Y -26.708,Z -64.398,A -90.000,B 90.000,C 0.000} C_DIS
LIN {X 78.964,Y -27.151,Z -64.478,A -90.000,B 90.000,C 0.000} C_DIS
LIN {X 79.079,Y -27.717,Z -64.635,A -90.000,B 90.000,C 0.000} C_DIS
LIN {X 79.189,Y -28.102,Z -64.787,A -90.000,B 90.000,C 0.000} C_DIS
LIN {X 79.296,Y -28.403,Z -64.933,A -90.000,B 90.000,C 0.000} C_DIS
LIN {X 79.499,Y -28.927,Z -65.211,A -90.000,B 90.000,C 0.000} C_DIS
LIN {X 79.687,Y -29.329,Z -65.470,A -90.000,B 90.000,C 0.000} C_DIS
LIN {X 79.862,Y -29.637,Z -65.708,A -90.000,B 90.000,C 0.000} C_DIS
LIN {X 80.242,Y -30.212,Z -66.221,A -90.000,B 90.000,C 0.000} C_DIS
LIN {X 80.246,Y -40.094,Z -66.227,A -90.000,B 90.000,C 0.000} C_DIS
LIN {X 80.259,Y -40.786,Z -66.244,A -90.000,B 90.000,C 0.000} C_DIS
LIN {X 80.275,Y -41.201,Z -66.266,A -90.000,B 90.000,C 0.000} C_DIS
LIN {X 80.308,Y -41.587,Z -66.310,A -90.000,B 90.000,C 0.000} C_DIS
LIN {X 80.372,Y -42.015,Z -66.394,A -90.000,B 90.000,C 0.000} C_DIS
LIN {X 80.432,Y -42.317,Z -66.473,A -90.000,B 90.000,C 0.000} C_DIS
LIN {X 80.545,Y -42.748,Z -66.619,A -90.000,B 90.000,C 0.000} C_DIS
LIN {X 80.646,Y -43.053,Z -66.746,A -90.000,B 90.000,C 0.000} C_DIS
LIN {X 80.736,Y -43.282,Z -66.857,A -90.000,B 90.000,C 0.000} C_DIS
LIN {X 80.853,Y -43.535,Z -66.990,A -90.000,B 90.000,C 0.000} C_DIS
LIN {X 80.887,Y -43.611,Z -67.026,A -90.000,B 90.000,C 0.000} C_DIS
LIN {X 80.949,Y -43.746,Z -67.086,A -90.000,B 90.000,C 0.000} C_DIS
LIN {X 81.001,Y -43.859,Z -67.129,A -90.000,B 90.000,C 0.000} C_DIS
LIN {X 81.045,Y -43.949,Z -67.157,A -90.000,B 90.000,C 0.000} C_DIS
LIN {X 81.063,Y -43.986,Z -67.165,A -90.000,B 90.000,C 0.000} C_DIS
LIN {X 81.080,Y -44.019,Z -67.169,A -90.000,B 90.000,C 0.000} C_DIS
LIN {X 81.095,Y -44.046,Z -67.169,A -90.000,B 90.000,C 0.000} C_DIS
LIN {X 81.109,Y -44.070,Z -67.166,A -90.000,B 90.000,C 0.000} C_DIS
LIN {X 81.120,Y -44.090,Z -67.158,A -90.000,B 90.000,C 0.000} C_DIS
LIN {X 81.130,Y -44.106,Z -67.147,A -90.000,B 90.000,C 0.000} C_DIS
LIN {X 81.138,Y -44.118,Z -67.133,A -90.000,B 90.000,C 0.000} C_DIS
LIN {X 81.144,Y -44.127,Z -67.114,A -90.000,B 90.000,C 0.000} C_DIS
LIN {X 81.149,Y -44.133,Z -67.092,A -90.000,B 90.000,C 0.000} C_DIS
LIN {X 81.152,Y -44.136,Z -67.067,A -90.000,B 90.000,C 0.000} C_DIS
LIN {X 81.154,Y -44.131,Z -67.006,A -90.000,B 90.000,C 0.000} C_DIS
LIN {X 81.154,Y -44.123,Z -66.970,A -90.000,B 90.000,C 0.000} C_DIS
LIN {X 81.151,Y -44.113,Z -66.930,A -90.000,B 90.000,C 0.000} C_DIS
LIN {X 81.143,Y -44.080,Z -66.841,A -90.000,B 90.000,C 0.000} C_DIS
LIN {X 81.131,Y -44.033,Z -66.740,A -90.000,B 90.000,C 0.000} C_DIS
LIN {X 81.094,Y -43.918,Z -66.497,A -90.000,B 90.000,C 0.000} C_DIS
LIN {X 81.045,Y -43.767,Z -66.206,A -90.000,B 90.000,C 0.000} C_DIS
LIN {X 80.987,Y -43.522,Z -65.868,A -90.000,B 90.000,C 0.000} C_DIS
LIN {X 80.956,Y -43.343,Z -65.682,A -90.000,B 90.000,C 0.000} C_DIS
LIN {X 80.924,Y -43.102,Z -65.486,A -90.000,B 90.000,C 0.000} C_DIS
LIN {X 80.891,Y -42.753,Z -65.279,A -90.000,B 90.000,C 0.000} C_DIS
LIN {X 80.875,Y -42.499,Z -65.172,A -90.000,B 90.000,C 0.000} C_DIS
LIN {X 80.858,Y -42.106,Z -65.062,A -90.000,B 90.000,C 0.000} C_DIS
LIN {X 80.850,Y -41.713,Z -65.006,A -90.000,B 90.000,C 0.000} C_DIS
LIN {X 80.844,Y -41.160,Z -64.964,A -90.000,B 90.000,C 0.000} C_DIS
LIN {X 80.842,Y -30.408,Z -64.950,A -90.000,B 90.000,C 0.000} C_DIS
LIN {X 80.795,Y -30.241,Z -64.599,A -90.000,B 90.000,C 0.000} C_DIS
LIN {X 80.736,Y -30.016,Z -64.098,A -90.000,B 90.000,C 0.000} C_DIS
LIN {X 80.710,Y -29.895,Z -63.835,A -90.000,B 90.000,C 0.000} C_DIS
LIN {X 80.686,Y -29.768,Z -63.564,A -90.000,B 90.000,C 0.000} C_DIS
LIN {X 80.666,Y -29.634,Z -63.284,A -90.000,B 90.000,C 0.000} C_DIS
LIN {X 80.649,Y -29.495,Z -62.997,A -90.000,B 90.000,C 0.000} C_DIS
LIN {X 80.636,Y -29.349,Z -62.702,A -90.000,B 90.000,C 0.000} C_DIS
LIN {X 80.627,Y -29.197,Z -62.401,A -90.000,B 90.000,C 0.000} C_DIS
LIN {X 80.625,Y -29.117,Z -62.247,A -90.000,B 90.000,C 0.000} C_DIS
LIN {X 80.623,Y -28.950,Z -61.935,A -90.000,B 90.000,C 0.000} C_DIS
LIN {X 80.628,Y -28.779,Z -61.617,A -90.000,B 90.000,C 0.000} C_DIS
LIN {X 80.638,Y -28.604,Z -61.293,A -90.000,B 90.000,C 0.000} C_DIS
LIN {X 80.655,Y -28.426,Z -60.963,A -90.000,B 90.000,C 0.000} C_DIS
LIN {X 80.678,Y -28.249,Z -60.627,A -90.000,B 90.000,C 0.000} C_DIS
LIN {X 80.693,Y -28.162,Z -60.458,A -90.000,B 90.000,C 0.000} C_DIS
LIN {X 80.728,Y -27.985,Z -60.115,A -90.000,B 90.000,C 0.000} C_DIS
LIN {X 80.748,Y -27.893,Z -59.942,A -90.000,B 90.000,C 0.000} C_DIS
LIN {X 80.770,Y -27.792,Z -59.767,A -90.000,B 90.000,C 0.000} C_DIS
LIN {X 80.795,Y -27.670,Z -59.592,A -90.000,B 90.000,C 0.000} C_DIS
LIN {X 80.821,Y -27.536,Z -59.415,A -90.000,B 90.000,C 0.000} C_DIS
LIN {X 80.850,Y -27.393,Z -59.238,A -90.000,B 90.000,C 0.000} C_DIS
LIN {X 80.881,Y -27.285,Z -59.059,A -90.000,B 90.000,C 0.000} C_DIS
LIN {X 80.951,Y -27.134,Z -58.699,A -90.000,B 90.000,C 0.000} C_DIS
LIN {X 80.989,Y -27.060,Z -58.518,A -90.000,B 90.000,C 0.000} C_DIS
LIN {X 81.073,Y -26.916,Z -58.153,A -90.000,B 90.000,C 0.000} C_DIS
LIN {X 81.119,Y -26.849,Z -57.969,A -90.000,B 90.000,C 0.000} C_DIS
LIN {X 81.167,Y -26.785,Z -57.785,A -90.000,B 90.000,C 0.000} C_DIS
LIN {X 81.219,Y -26.726,Z -57.600,A -90.000,B 90.000,C 0.000} C_DIS
LIN {X 81.273,Y -26.672,Z -57.414,A -90.000,B 90.000,C 0.000} C_DIS
LIN {X 81.329,Y -26.595,Z -57.228,A -90.000,B 90.000,C 0.000} C_DIS
LIN {X 81.389,Y -26.491,Z -57.041,A -90.000,B 90.000,C 0.000} C_DIS
LIN {X 81.517,Y -26.272,Z -56.666,A -90.000,B 90.000,C 0.000} C_DIS
LIN {X 81.586,Y -26.155,Z -56.478,A -90.000,B 90.000,C 0.000} C_DIS
LIN {X 81.658,Y -26.025,Z -56.289,A -90.000,B 90.000,C 0.000} C_DIS
LIN {X 81.733,Y -23.308,Z -56.100,A -90.000,B 90.000,C 0.000} C_DIS
LIN {X 82.012,Y -23.308,Z -55.411,A -90.000,B 90.000,C 0.000} C_DIS
LIN {X 82.012,Y -60.000,Z -55.411,A -90.000,B 90.000,C 0.000} C_DIS
LIN {X 103.228,Y -60.000,Z -37.495,A -90.000,B 90.000,C 0.000} C_DIS
LIN {X 103.228,Y -23.308,Z -37.495,A -90.000,B 90.000,C 0.000} C_DIS
LIN {X 103.314,Y -23.308,Z -37.457,A -90.000,B 90.000,C 0.000} C_DIS
LIN {X 103.314,Y -60.000,Z -37.457,A -90.000,B 90.000,C 0.000} C_DIS
LIN {X 117.350,Y -60.000,Z -45.336,A -90.000,B 90.000,C 0.000} C_DIS
LIN {X 117.350,Y -23.308,Z -45.336,A -90.000,B 90.000,C 0.000} C_DIS
LIN {X 117.260,Y -23.308,Z -45.739,A -90.000,B 90.000,C 0.000} C_DIS
LIN {X 117.243,Y -23.308,Z -45.810,A -90.000,B 90.000,C 0.000} C_DIS
LIN {X 117.248,Y -23.307,Z -45.816,A -90.000,B 90.000,C 0.000} C_DIS
LIN {X 117.239,Y -23.308,Z -45.841,A -90.000,B 90.000,C 0.000} C_DIS
LIN {X 117.219,Y -23.308,Z -45.879,A -90.000,B 90.000,C 0.000} C_DIS
LIN {X 117.211,Y -23.308,Z -45.903,A -90.000,B 90.000,C 0.000} C_DIS
LIN {X 117.211,Y -60.000,Z -45.903,A -90.000,B 90.000,C 0.000} C_DIS
LIN {X 99.738,Y -60.000,Z -85.770,A -90.000,B 90.000,C 0.000} C_DIS
LIN {X 99.738,Y -23.308,Z -85.770,A -90.000,B 90.000,C 0.000} C_DIS
LIN {X 99.783,Y -23.308,Z -86.350,A -90.000,B 90.000,C 0.000} C_DIS
LIN {X 99.783,Y -60.000,Z -86.350,A -90.000,B 90.000,C 0.000} C_DIS
LIN {X 12.457,Y -60.000,Z -49.463,A -90.000,B 90.000,C 0.000} C_DIS
LIN {X 12.457,Y -23.308,Z -49.463,A -90.000,B 90.000,C 0.000} C_DIS
LIN {X 12.861,Y -23.430,Z -49.538,A -90.000,B 90.000,C 0.000} C_DIS
LIN {X 12.912,Y -23.446,Z -49.548,A -90.000,B 90.000,C 0.000} C_DIS
LIN {X 13.069,Y -23.484,Z -49.523,A -90.000,B 90.000,C 0.000} C_DIS
LIN {X 13.279,Y -23.536,Z -49.490,A -90.000,B 90.000,C 0.000} C_DIS
LIN {X 13.427,Y -23.571,Z -49.471,A -90.000,B 90.000,C 0.000} C_DIS
LIN {X 13.577,Y -23.606,Z -49.458,A -90.000,B 90.000,C 0.000} C_DIS
LIN {X 13.698,Y -23.599,Z -49.301,A -90.000,B 90.000,C 0.000} C_DIS
LIN {X 13.924,Y -23.566,Z -49.030,A -90.000,B 90.000,C 0.000} C_DIS
LIN {X 13.999,Y -23.555,Z -48.943,A -90.000,B 90.000,C 0.000} C_DIS
LIN {X 14.065,Y -23.547,Z -48.871,A -90.000,B 90.000,C 0.000} C_DIS
LIN {X 14.119,Y -23.544,Z -48.808,A -90.000,B 90.000,C 0.000} C_DIS
LIN {X 14.220,Y -23.541,Z -48.700,A -90.000,B 90.000,C 0.000} C_DIS
LIN {X 14.345,Y -23.538,Z -48.578,A -90.000,B 90.000,C 0.000} C_DIS
LIN {X 14.497,Y -23.531,Z -48.431,A -90.000,B 90.000,C 0.000} C_DIS
LIN {X 14.559,Y -23.524,Z -48.375,A -90.000,B 90.000,C 0.000} C_DIS
LIN {X 14.711,Y -23.521,Z -48.228,A -90.000,B 90.000,C 0.000} C_DIS
LIN {X 15.047,Y -23.505,Z -47.913,A -90.000,B 90.000,C 0.000} C_DIS
LIN {X 15.280,Y -23.484,Z -47.718,A -90.000,B 90.000,C 0.000} C_DIS
LIN {X 15.560,Y -23.449,Z -47.491,A -90.000,B 90.000,C 0.000} C_DIS
LIN {X 15.709,Y -23.439,Z -47.369,A -90.000,B 90.000,C 0.000} C_DIS
LIN {X 15.747,Y -23.436,Z -47.339,A -90.000,B 90.000,C 0.000} C_DIS
LIN {X 15.856,Y -23.430,Z -47.256,A -90.000,B 90.000,C 0.000} C_DIS
LIN {X 15.947,Y -23.426,Z -47.191,A -90.000,B 90.000,C 0.000} C_DIS
LIN {X 16.166,Y -23.399,Z -47.043,A -90.000,B 90.000,C 0.000} C_DIS
LIN {X 16.592,Y -23.333,Z -46.763,A -90.000,B 90.000,C 0.000} C_DIS
LIN {X 16.765,Y -23.308,Z -46.654,A -90.000,B 90.000,C 0.000} C_DIS
LIN {X 16.765,Y -60.000,Z -46.654,A -90.000,B 90.000,C 0.000} C_DIS
LIN {X -32.429,Y -60.000,Z -47.782,A -90.000,B 90.000,C 0.000} C_DIS
LIN {X -32.429,Y -23.308,Z -47.782,A -90.000,B 90.000,C 0.000} C_DIS
LIN {X -32.019,Y -23.340,Z -47.873,A -90.000,B 90.000,C 0.000} C_DIS
LIN {X -31.859,Y -23.351,Z -47.911,A -90.000,B 90.000,C 0.000} C_DIS
LIN {X -31.266,Y -23.388,Z -48.059,A -90.000,B 90.000,C 0.000} C_DIS
LIN {X -30.126,Y -23.451,Z -48.352,A -90.000,B 90.000,C 0.000} C_DIS
LIN {X -29.193,Y -23.499,Z -48.596,A -90.000,B 90.000,C 0.000} C_DIS
LIN {X -28.512,Y -23.532,Z -48.781,A -90.000,B 90.000,C 0.000} C_DIS
LIN {X -27.376,Y -23.583,Z -49.105,A -90.000,B 90.000,C 0.000} C_DIS
LIN {X -27.020,Y -23.596,Z -49.207,A -90.000,B 90.000,C 0.000} C_DIS
LIN {X -26.413,Y -23.627,Z -49.379,A -90.000,B 90.000,C 0.000} C_DIS
LIN {X -25.344,Y -23.683,Z -49.669,A -90.000,B 90.000,C 0.000} C_DIS
LIN {X -24.500,Y -23.726,Z -49.903,A -90.000,B 90.000,C 0.000} C_DIS
LIN {X -24.239,Y -23.741,Z -49.973,A -90.000,B 90.000,C 0.000} C_DIS
LIN {X -23.185,Y -23.798,Z -50.241,A -90.000,B 90.000,C 0.000} C_DIS
LIN {X -22.725,Y -23.826,Z -50.368,A -90.000,B 90.000,C 0.000} C_DIS
LIN {X -22.537,Y -23.838,Z -50.410,A -90.000,B 90.000,C 0.000} C_DIS
LIN {X -22.273,Y -23.855,Z -50.466,A -90.000,B 90.000,C 0.000} C_DIS
LIN {X -21.935,Y -23.876,Z -50.533,A -90.000,B 90.000,C 0.000} C_DIS
LIN {X -21.590,Y -23.898,Z -50.608,A -90.000,B 90.000,C 0.000} C_DIS
LIN {X -20.995,Y -23.940,Z -50.676,A -90.000,B 90.000,C 0.000} C_DIS
LIN {X -20.771,Y -23.961,Z -50.589,A -90.000,B 90.000,C 0.000} C_DIS
LIN {X -20.680,Y -23.969,Z -50.556,A -90.000,B 90.000,C 0.000} C_DIS
LIN {X -20.530,Y -23.981,Z -50.506,A -90.000,B 90.000,C 0.000} C_DIS
LIN {X -20.234,Y -24.007,Z -50.362,A -90.000,B 90.000,C 0.000} C_DIS
LIN {X -19.796,Y -24.046,Z -50.168,A -90.000,B 90.000,C 0.000} C_DIS
LIN {X -19.479,Y -24.074,Z -50.011,A -90.000,B 90.000,C 0.000} C_DIS
LIN {X -19.088,Y -24.108,Z -49.832,A -90.000,B 90.000,C 0.000} C_DIS
LIN {X -18.875,Y -24.128,Z -49.736,A -90.000,B 90.000,C 0.000} C_DIS
LIN {X -18.526,Y -24.160,Z -49.581,A -90.000,B 90.000,C 0.000} C_DIS
LIN {X -17.998,Y -24.194,Z -49.360,A -90.000,B 90.000,C 0.000} C_DIS
LIN {X -17.805,Y -24.202,Z -49.283,A -90.000,B 90.000,C 0.000} C_DIS
LIN {X -17.222,Y -24.223,Z -49.061,A -90.000,B 90.000,C 0.000} C_DIS
LIN {X -16.981,Y -24.227,Z -48.970,A -90.000,B 90.000,C 0.000} C_DIS
LIN {X -16.569,Y -24.234,Z -48.825,A -90.000,B 90.000,C 0.000} C_DIS
LIN {X -16.371,Y -24.236,Z -48.762,A -90.000,B 90.000,C 0.000} C_DIS
LIN {X -16.145,Y -24.241,Z -48.701,A -90.000,B 90.000,C 0.000} C_DIS
LIN {X -15.994,Y -24.245,Z -48.664,A -90.000,B 90.000,C 0.000} C_DIS
